// TwinCAT 3 PLC project PLC_TMO_VAC
// Title: lcls-plc-tmo-vac
// Company: SLAC
// ProjectVersion: 0.0.0
// ProgramVersion: 3.1.4022.7
// libraries:
//   LCLS General, * (SLAC)
//   LCLS Vacuum, * (SLAC - LCLS)
//   LCLSVacuumSerialDriverLib, * (SLAC - LCLS)
//   PMPS, * (SLAC - LCLS)
//   Tc2_SerialCom, * (Beckhoff Automation GmbH)
//   Tc2_Standard, * (Beckhoff Automation GmbH)
//   Tc2_System, * (Beckhoff Automation GmbH)
//   Tc3_Module, * (Beckhoff Automation GmbH)
// project tree:
//   / ComTask.TcTTO (not stored), FSVTask.TcTTO (not stored), PlcTask.TcTTO (not stored)
//   DUTs/ E_STATES.TcDUT (not stored)
//   GVLs/ GVL_COM.TcGVL (not stored), GVL_FEE_Device.TcGVL (not stored), GVL_FSV_PMPS.TcGVL, GVL_FS_Devices.TcGVL (not stored), GVL_Hutch_Gauges.TcGVL (not stored), GVL_Hutch_Pumps.TcGVL (not stored), GVL_Hutch_Valves.TcGVL (not stored), GVL_IP1_ECAT.TcGVL (not stored), GVL_PMPS.TcGVL, GVL_Variables.TcGVL
//   POUs/ DIAGNOSTICS.TcPOU (not stored), FB_VRC_NO_FFO_VLS.TcPOU (not stored), F_Turbo_Protection_ILK.TcPOU (not stored), MAIN.TcPOU, PRG_HV_SAFETY.TcPOU (not stored), PRG_PMPS.TcPOU, PRG_Hutch_Ion_Pumps.TcPOU (not stored), PRG_COM.TcPOU (not stored), PRG_FEE.TcPOU (not stored), PRG_FSV.TcPOU (not stored), PRG_FSV_Interfaces.TcPOU (not stored), PRG_Hutch_Beamline_Valves.TcPOU, PRG_Hutch_Gauges.TcPOU (not stored), PRG_IP1_ECAT_Interfaces.TcPOU (not stored), PRG_Roughing_Pumps.TcPOU, PRG_Section_2.TcPOU (not stored)
// real-time tasks:
//   TASK PlcTask: cycle T#10ms, priority 20, ADS port 350
//   TASK ComTask: cycle T#11ms, priority 30, ADS port 351
//   TASK FSVTask: cycle T#2ms, priority 15, ADS port 352
// I/O:
//   DEVICE Device 1 (EtherCAT)
// variable links:
//   PLC_TMO_VAC Instance <-> Device 1 (EtherCAT)/B940-R20-CX0 (EK1200)/CX0_E1 (EL2202)
//     ComTask Outputs/GVL_PMPS.g_FastFaultOutput1.q_xFastFaultOut <-> Channel 1/Output
//     ComTask Outputs/GVL_PMPS.g_FastFaultOutput2.q_xFastFaultOut <-> Channel 2/Output
//   PLC_TMO_VAC Instance <-> Device 1 (EtherCAT)/B940-R20-CX0 (EK1200)/CX0_E10_QPC2 (EL1004)
//     ComTask Inputs/GVL_FEE_Device.PC4K4_XTES_PIP_01.i_xSP_DI <-> Channel 1/Input
//     ComTask Inputs/GVL_FEE_Device.TV1K4_PIP_01.i_xSP_DI <-> Channel 3/Input
//     ComTask Inputs/GVL_Hutch_Pumps.MR2K4_KBO_PIP_01.i_xSP_DI <-> Channel 2/Input
//     ComTask Inputs/GVL_Hutch_Pumps.MR4K4_KBO_PIP_01.i_xSP_DI <-> Channel 4/Input
//   PLC_TMO_VAC Instance <-> Device 1 (EtherCAT)/B940-R20-CX0 (EK1200)/CX0_E11_QPC2 (EL2794)
//     ComTask Outputs/GVL_FEE_Device.PC4K4_XTES_PIP_01.q_xHVEna_DO <-> Channel 1/Output
//     ComTask Outputs/GVL_FEE_Device.TV1K4_PIP_01.q_xHVEna_DO <-> Channel 3/Output
//     ComTask Outputs/GVL_Hutch_Pumps.MR2K4_KBO_PIP_01.q_xHVEna_DO <-> Channel 2/Output
//     ComTask Outputs/GVL_Hutch_Pumps.MR4K4_KBO_PIP_01.q_xHVEna_DO <-> Channel 4/Output
//   PLC_TMO_VAC Instance <-> Device 1 (EtherCAT)/B940-R20-CX0 (EK1200)/CX0_E13 (EK1122)/IP1_ECAT (EL6692)
//     ComTask Inputs/GVL_IP1_ECAT.IP1_HV_SAFETY_ENABLE <-> IO Inputs/IP1_HV_SAFETY_ENABLE
//     ComTask Inputs/GVL_IP1_ECAT.IP1_MAIN_GAUGE.i_rPRESS <-> IO Inputs/IP1_MAIN_rPRESS
//     ComTask Inputs/GVL_IP1_ECAT.IP1_MAIN_GAUGE.i_xAT_VAC <-> IO Inputs/IP1_MAIN_xAT_VAC
//     ComTask Inputs/GVL_IP1_ECAT.IP1_MAIN_GAUGE.i_xPRESS_OK <-> IO Inputs/IP1_MAIN_xPRESS_OK
//     ComTask Inputs/GVL_IP1_ECAT.IP1_PLC_NAME <-> IO Inputs/ENDSTATION_PLC_NAME
//     ComTask Inputs/GVL_IP1_ECAT.IP1_ROUGH_VRC_01_AtOpnLS <-> IO Inputs/IP1_ROUGH_VRC_01_OPEN_LS
//     ComTask Inputs/GVL_IP1_ECAT.IP1_ROUGH_VRC_02_AtOpnLS <-> IO Inputs/IP1_ROUGH_VRC_02_OPEN_LS
//     ComTask Inputs/GVL_IP1_ECAT.IP1_ROUGH_VRC_03_AtOpnLS <-> IO Inputs/IP1_ROUGH_VRC_03_OPEN_LS
//     ComTask Inputs/GVL_IP1_ECAT.IP1_TURBOS_ALL_AtSpd <-> IO Inputs/IP1_TURBOS_ALL_AtSpd
//     ComTask Inputs/GVL_IP1_ECAT.xEcatBridge_External_device_not_connected <-> SYNC Inputs/External device not connected
//     ComTask Inputs/GVL_IP1_ECAT.xEcatBridge_TxPDO_state <-> SYNC Inputs/TxPDO state
//     ComTask Inputs/GVL_IP1_ECAT.xEcatBridge_WcState <-> WcState/WcState
//     ComTask Outputs/GVL_IP1_ECAT.My_PLC_NAME <-> IO Outputs/HUTCH_PLC_NAME
//     ComTask Outputs/GVL_IP1_ECAT.ROUGH1_VRC_01_AtOpnLS <-> IO Outputs/TMO_ROUGH1_VRC_01_OPEN_LS
//     ComTask Outputs/GVL_IP1_ECAT.ROUGH2_VRC_01_AtOpnLS <-> IO Outputs/TMO_ROUGH2_VRC_01_OPEN_LS
//   PLC_TMO_VAC Instance <-> Device 1 (EtherCAT)/B940-R20-CX0 (EK1200)/CX0_E1A (EL2202)
//     FSVTask Outputs/GVL_PMPS.g_FastFaultOutput3.q_xFastFaultOut <-> Channel 1/Output
//     FSVTask Outputs/GVL_PMPS.g_FastFaultOutput4.q_xFastFaultOut <-> Channel 2/Output
//   PLC_TMO_VAC Instance <-> Device 1 (EtherCAT)/B940-R20-CX0 (EK1200)/CX0_E2_EXILK (EL1008)
//     ComTask Inputs/GVL_FEE_Device.USVacOk_HI <-> Channel 1/Input
//     ComTask Inputs/GVL_FEE_Device.USVacOk_LO <-> Channel 3/Input
//   PLC_TMO_VAC Instance <-> Device 1 (EtherCAT)/B940-R20-CX0 (EK1200)/CX0_E6_QPC1 (EL3064)
//     ComTask Inputs/GVL_FEE_Device.MR1K4_SOMS_PIP_01.i_iPRESS <-> AI Standard Channel 1/Value
//     ComTask Inputs/GVL_FEE_Device.ST1K4_TEST_PIP_01.i_iPRESS <-> AI Standard Channel 2/Value
//     ComTask Inputs/GVL_FEE_Device.ST2K4_BCS_PIP_01.i_iPRESS <-> AI Standard Channel 3/Value
//     ComTask Inputs/GVL_FEE_Device.ST3K4_PPS_PIP_01.i_iPRESS <-> AI Standard Channel 4/Value
//   PLC_TMO_VAC Instance <-> Device 1 (EtherCAT)/B940-R20-CX0 (EK1200)/CX0_E7_QPC1 (EL1004)
//     ComTask Inputs/GVL_FEE_Device.MR1K4_SOMS_PIP_01.i_xSP_DI <-> Channel 1/Input
//     ComTask Inputs/GVL_FEE_Device.ST1K4_TEST_PIP_01.i_xSP_DI <-> Channel 2/Input
//     ComTask Inputs/GVL_FEE_Device.ST2K4_BCS_PIP_01.i_xSP_DI <-> Channel 3/Input
//     ComTask Inputs/GVL_FEE_Device.ST3K4_PPS_PIP_01.i_xSP_DI <-> Channel 4/Input
//   PLC_TMO_VAC Instance <-> Device 1 (EtherCAT)/B940-R20-CX0 (EK1200)/CX0_E8_QPC1 (EL2794)
//     ComTask Outputs/GVL_FEE_Device.MR1K4_SOMS_PIP_01.q_xHVEna_DO <-> Channel 1/Output
//     ComTask Outputs/GVL_FEE_Device.ST1K4_TEST_PIP_01.q_xHVEna_DO <-> Channel 2/Output
//     ComTask Outputs/GVL_FEE_Device.ST2K4_BCS_PIP_01.q_xHVEna_DO <-> Channel 3/Output
//     ComTask Outputs/GVL_FEE_Device.ST3K4_PPS_PIP_01.q_xHVEna_DO <-> Channel 4/Output
//   PLC_TMO_VAC Instance <-> Device 1 (EtherCAT)/B940-R20-CX0 (EK1200)/CX0_E9_QPC2 (EL3064)
//     ComTask Inputs/GVL_FEE_Device.PC4K4_XTES_PIP_01.i_iPRESS <-> AI Standard Channel 1/Value
//     ComTask Inputs/GVL_FEE_Device.TV1K4_PIP_01.i_iPRESS <-> AI Standard Channel 3/Value
//     ComTask Inputs/GVL_Hutch_Pumps.MR2K4_KBO_PIP_01.i_iPRESS <-> AI Standard Channel 2/Value
//     ComTask Inputs/GVL_Hutch_Pumps.MR4K4_KBO_PIP_01.i_iPRESS <-> AI Standard Channel 4/Value
//   PLC_TMO_VAC Instance <-> Device 1 (EtherCAT)/B940_K4S20_EB1  (EP2338-0002)
//     ComTask Inputs/GVL_FEE_Device.TV1K4_VGC_01.i_xClsLS <-> Channel 2/Input
//     ComTask Inputs/GVL_FEE_Device.TV1K4_VGC_02.i_xClsLS <-> Channel 6/Input
//     ComTask Inputs/GVL_FEE_Device.TV1K4_VGC_01.i_xOpnLS <-> Channel 1/Input
//     ComTask Inputs/GVL_FEE_Device.TV1K4_VGC_02.i_xOpnLS <-> Channel 5/Input
//     ComTask Outputs/GVL_FEE_Device.TV1K4_VGC_01.q_xOPN_DO <-> Channel 11/Output
//     ComTask Outputs/GVL_FEE_Device.TV1K4_VGC_02.q_xOPN_DO <-> Channel 15/Output
//   PLC_TMO_VAC Instance <-> Device 1 (EtherCAT)/B940_K4S20_EB2  (EP3174-0002)
//     ComTask Inputs/GVL_FEE_Device.TV1K4_GCC_01.i_iPRESS_R <-> AI Standard Channel 2/Value
//     ComTask Inputs/GVL_FEE_Device.TV1K4_GPI_01.i_iPRESS_R <-> AI Standard Channel 1/Value
//   PLC_TMO_VAC Instance <-> Device 1 (EtherCAT)/B940_K4S20_EB3 (EP2624-0002)
//     ComTask Outputs/GVL_FEE_Device.TV1K4_GCC_01.q_xHV_DIS <-> Channel 1/Output
//   PLC_TMO_VAC Instance <-> Device 1 (EtherCAT)/B940_K4S20_EK0  (EK1100)/K4S20-E1-FSV (EL1004)
//     FSVTask Inputs/GVL_FS_Devices.TV1K4_VFS_1.i_xClsLS <-> Channel 1/Input
//     FSVTask Inputs/GVL_FS_Devices.TV1K4_VFS_1.i_xOpnLS <-> Channel 2/Input
//   PLC_TMO_VAC Instance <-> Device 1 (EtherCAT)/B940_K4S20_EK0  (EK1100)/K4S20-E2-FSV (EL2202)
//     FSVTask Outputs/GVL_FS_Devices.TV1K4_VFS_1.q_xClose_A <-> Channel 1/Output
//     FSVTask Outputs/GVL_FS_Devices.TV1K4_VFS_1.q_xClose_B <-> Channel 2/Output
//   PLC_TMO_VAC Instance <-> Device 1 (EtherCAT)/B940_K4S20_EK0  (EK1100)/K4S20-E3-FSV (EL2202)
//     FSVTask Outputs/GVL_FS_Devices.TV1K4_VFS_1.q_xClose_C <-> Channel 1/Output
//     FSVTask Outputs/GVL_FS_Devices.TV1K4_VFS_1.q_xOPN_DO <-> Channel 2/Output
//   PLC_TMO_VAC Instance <-> Device 1 (EtherCAT)/B940_K4S24_EB1 (EP3174-0002)
//     ComTask Inputs/GVL_FEE_Device.ST1K4_TEST_GCC_01.i_iPRESS_R <-> AI Standard Channel 2/Value
//     ComTask Inputs/GVL_FEE_Device.ST1K4_TEST_GPI_01.i_iPRESS_R <-> AI Standard Channel 1/Value
//   PLC_TMO_VAC Instance <-> Device 1 (EtherCAT)/B940_K4S24_EB2 (EP2624-0002)
//     ComTask Outputs/GVL_FEE_Device.ST1K4_TEST_GCC_01.q_xHV_DIS <-> Channel 1/Output
//   PLC_TMO_VAC Instance <-> Device 1 (EtherCAT)/B940_K4S28_EB1 (EP3174-0002)
//     ComTask Inputs/GVL_FEE_Device.ST2K4_BCS_GCC_01.i_iPRESS_R <-> AI Standard Channel 2/Value
//     ComTask Inputs/GVL_FEE_Device.ST2K4_BCS_GPI_01.i_iPRESS_R <-> AI Standard Channel 1/Value
//   PLC_TMO_VAC Instance <-> Device 1 (EtherCAT)/B940_K4S28_EB2 (EP2624-0002)
//     ComTask Outputs/GVL_FEE_Device.ST2K4_BCS_GCC_01.q_xHV_DIS <-> Channel 1/Output
//   PLC_TMO_VAC Instance <-> Device 1 (EtherCAT)/B940_K4S33_EB1 (EP2338-0002)
//     ComTask Inputs/GVL_FEE_Device.ST3K4_PPS_VGC_01.i_xClsLS <-> Channel 2/Input
//     ComTask Inputs/GVL_FEE_Device.ST3K4_PPS_VGC_01.i_xOpnLS <-> Channel 1/Input
//     ComTask Outputs/GVL_FEE_Device.ST3K4_PPS_VGC_01.q_xOPN_DO <-> Channel 11/Output
//   PLC_TMO_VAC Instance <-> Device 1 (EtherCAT)/B940_K4S33_EB2 (EP3174-0002)
//     ComTask Inputs/GVL_FEE_Device.PC4K4_XTES_GCC_01.i_iPRESS_R <-> AI Standard Channel 2/Value
//     ComTask Inputs/GVL_FEE_Device.PC4K4_XTES_GPI_01.i_iPRESS_R <-> AI Standard Channel 1/Value
//   PLC_TMO_VAC Instance <-> Device 1 (EtherCAT)/B940_K4S33_EB3 (EP2624-0002)
//     ComTask Outputs/GVL_FEE_Device.PC4K4_XTES_GCC_01.q_xHV_DIS <-> Channel 1/Output
//   PLC_TMO_VAC Instance <-> Device 1 (EtherCAT)/B940_R20_EK0 (EK1100)/R20_EK0_E1_MKS937B (EL3064)
//     ComTask Inputs/GVL_Hutch_Gauges.LI2K4_IP1_GFS_01.i_iPRESS_R <-> AI Standard Channel 1/Value
//   PLC_TMO_VAC Instance <-> Device 1 (EtherCAT)/B940_R20_EK0 (EK1100)/R20_EK0_E3_MKS937B (EL2794)
//     ComTask Outputs/GVL_Hutch_Gauges.LI2K4_IP1_GFS_01.q_xHV_DIS <-> Channel 1/Output
//     ComTask Outputs/GVL_Hutch_Pumps.PA2K4_IP1_PIP_01.q_xHVEna_DO <-> Channel 4/Output
//   PLC_TMO_VAC Instance <-> Device 1 (EtherCAT)/B940_R20_EK0 (EK1100)/R20_EK0_E5_MKS937B (EL1124)
//     ComTask Inputs/GVL_Hutch_Pumps.PA2K4_IP1_PIP_01.i_xError <-> Channel 4/Input
//     ComTask Inputs/GVL_Hutch_Pumps.PA2K4_IP1_PIP_01.i_xIP_ON <-> Channel 3/Input
//     FSVTask Inputs/GVL_FS_Devices.MR3K4_KBO_VFS_1.i_xTrigger <-> Channel 1/Input
//     FSVTask Inputs/GVL_FS_Devices.MR4K4_KBO_VFS_1.i_xTrigger <-> Channel 1/Input
//     FSVTask Inputs/GVL_FS_Devices.TV1K4_VFS_1.i_xTrigger <-> Channel 1/Input
//   PLC_TMO_VAC Instance <-> Device 1 (EtherCAT)/B940_R20_EK0 (EK1100)/R20_EK0_SIP (EL3174-0002)
//     ComTask Inputs/GVL_Hutch_Pumps.PA2K4_IP1_PIP_01.i_iPRESS <-> AI Standard Channel 1/Value
//   PLC_TMO_VAC Instance <-> Device 1 (EtherCAT)/TMO_K4S2_ EP1 (EP4374-0002)
//     ComTask Inputs/GVL_Hutch_Gauges.TMO_ROUGH1_GPI_02.i_iPRESS_R <-> AI Inputs Channel 1/Value
//     ComTask Inputs/GVL_Hutch_Gauges.TMO_ROUGH2_GPI_02.i_iPRESS_R <-> AI Inputs Channel 2/Value
//     ComTask Outputs/GVL_Hutch_Valves.TMO_ROUGH1_VFV_02.q_iRawPosition <-> AO Outputs Channel 3/Analog output
//     ComTask Outputs/GVL_Hutch_Valves.TMO_ROUGH2_VFV_01.q_iRawPosition <-> AO Outputs Channel 4/Analog output
//   PLC_TMO_VAC Instance <-> Device 1 (EtherCAT)/TMO_K4S2_DRL_01 (EK1100)/K4S2_01_E1_VFS (EL1004)
//     FSVTask Inputs/GVL_FS_Devices.MR3K4_KBO_VFS_1.i_xClsLS <-> Channel 1/Input
//     FSVTask Inputs/GVL_FS_Devices.MR3K4_KBO_VFS_1.i_xOpnLS <-> Channel 2/Input
//   PLC_TMO_VAC Instance <-> Device 1 (EtherCAT)/TMO_K4S2_DRL_01 (EK1100)/K4S2_01_E3_VFS (EL2202)
//     FSVTask Outputs/GVL_FS_Devices.MR3K4_KBO_VFS_1.q_xClose_A <-> Channel 1/Output
//     FSVTask Outputs/GVL_FS_Devices.MR3K4_KBO_VFS_1.q_xClose_B <-> Channel 2/Output
//   PLC_TMO_VAC Instance <-> Device 1 (EtherCAT)/TMO_K4S2_DRL_01 (EK1100)/K4S2_01_E4_VFS (EL2202)
//     FSVTask Outputs/GVL_FS_Devices.MR3K4_KBO_VFS_1.q_xClose_C <-> Channel 1/Output
//     FSVTask Outputs/GVL_FS_Devices.MR3K4_KBO_VFS_1.q_xOPN_DO <-> Channel 2/Output
//   PLC_TMO_VAC Instance <-> Device 1 (EtherCAT)/TMO_K4S2_DRL_01 (EK1100)/K4S2_01_E5 (EL1004)
//     ComTask Inputs/GVL_Hutch_Valves.MR2K4_KBO_VWC_01.i_xClsLS <-> Channel 2/Input
//     ComTask Inputs/GVL_Hutch_Valves.MR3K4_KBO_VWC_01.i_xClsLS <-> Channel 4/Input
//     ComTask Inputs/GVL_Hutch_Valves.MR2K4_KBO_VWC_01.i_xOpnLS <-> Channel 1/Input
//     ComTask Inputs/GVL_Hutch_Valves.MR3K4_KBO_VWC_01.i_xOpnLS <-> Channel 3/Input
//   PLC_TMO_VAC Instance <-> Device 1 (EtherCAT)/TMO_K4S2_DRL_01 (EK1100)/K4S2_01_E6 (EL2004)
//     ComTask Outputs/GVL_Hutch_Valves.MR2K4_KBO_VWC_01.q_xOPN_DO <-> Channel 1/Output
//     ComTask Outputs/GVL_Hutch_Valves.MR3K4_KBO_VWC_01.q_xOPN_DO <-> Channel 2/Output
//   PLC_TMO_VAC Instance <-> Device 1 (EtherCAT)/TMO_K4S2_DRL_02 (EK1100)/K4S2_02_E1 (EL3174)
//     ComTask Inputs/GVL_Hutch_Gauges.MR2K4_KBO_GCC_01.i_iPRESS_R <-> AI Standard Channel 3/Value
//     ComTask Inputs/GVL_Hutch_Gauges.MR2K4_KBO_GPI_01.i_iPRESS_R <-> AI Standard Channel 2/Value
//     ComTask Inputs/GVL_Hutch_Gauges.PA1K4_IP1_GCC_01.i_iPRESS_R <-> AI Standard Channel 4/Value
//   PLC_TMO_VAC Instance <-> Device 1 (EtherCAT)/TMO_K4S2_DRL_02 (EK1100)/K4S2_02_E10 (EL6021)
//     ComTask Inputs/GVL_COM.K4S2_02_E10_stComIn/D[0] <-> COM TxPDO-Map Inputs/Data In 0
//     ComTask Inputs/GVL_COM.K4S2_02_E10_stComIn/D[10] <-> COM TxPDO-Map Inputs/Data In 10
//     ComTask Inputs/GVL_COM.K4S2_02_E10_stComIn/D[11] <-> COM TxPDO-Map Inputs/Data In 11
//     ComTask Inputs/GVL_COM.K4S2_02_E10_stComIn/D[12] <-> COM TxPDO-Map Inputs/Data In 12
//     ComTask Inputs/GVL_COM.K4S2_02_E10_stComIn/D[13] <-> COM TxPDO-Map Inputs/Data In 13
//     ComTask Inputs/GVL_COM.K4S2_02_E10_stComIn/D[14] <-> COM TxPDO-Map Inputs/Data In 14
//     ComTask Inputs/GVL_COM.K4S2_02_E10_stComIn/D[15] <-> COM TxPDO-Map Inputs/Data In 15
//     ComTask Inputs/GVL_COM.K4S2_02_E10_stComIn/D[16] <-> COM TxPDO-Map Inputs/Data In 16
//     ComTask Inputs/GVL_COM.K4S2_02_E10_stComIn/D[17] <-> COM TxPDO-Map Inputs/Data In 17
//     ComTask Inputs/GVL_COM.K4S2_02_E10_stComIn/D[18] <-> COM TxPDO-Map Inputs/Data In 18
//     ComTask Inputs/GVL_COM.K4S2_02_E10_stComIn/D[19] <-> COM TxPDO-Map Inputs/Data In 19
//     ComTask Inputs/GVL_COM.K4S2_02_E10_stComIn/D[1] <-> COM TxPDO-Map Inputs/Data In 1
//     ComTask Inputs/GVL_COM.K4S2_02_E10_stComIn/D[20] <-> COM TxPDO-Map Inputs/Data In 20
//     ComTask Inputs/GVL_COM.K4S2_02_E10_stComIn/D[21] <-> COM TxPDO-Map Inputs/Data In 21
//     ComTask Inputs/GVL_COM.K4S2_02_E10_stComIn/D[2] <-> COM TxPDO-Map Inputs/Data In 2
//     ComTask Inputs/GVL_COM.K4S2_02_E10_stComIn/D[3] <-> COM TxPDO-Map Inputs/Data In 3
//     ComTask Inputs/GVL_COM.K4S2_02_E10_stComIn/D[4] <-> COM TxPDO-Map Inputs/Data In 4
//     ComTask Inputs/GVL_COM.K4S2_02_E10_stComIn/D[5] <-> COM TxPDO-Map Inputs/Data In 5
//     ComTask Inputs/GVL_COM.K4S2_02_E10_stComIn/D[6] <-> COM TxPDO-Map Inputs/Data In 6
//     ComTask Inputs/GVL_COM.K4S2_02_E10_stComIn/D[7] <-> COM TxPDO-Map Inputs/Data In 7
//     ComTask Inputs/GVL_COM.K4S2_02_E10_stComIn/D[8] <-> COM TxPDO-Map Inputs/Data In 8
//     ComTask Inputs/GVL_COM.K4S2_02_E10_stComIn/D[9] <-> COM TxPDO-Map Inputs/Data In 9
//     ComTask Inputs/GVL_COM.K4S2_02_E10_stComIn/Status <-> COM TxPDO-Map Inputs/Status
//     ComTask Outputs/GVL_COM.K4S2_02_E10_stComOut/Ctrl <-> COM RxPDO-Map Outputs/Ctrl
//     ComTask Outputs/GVL_COM.K4S2_02_E10_stComOut/D[0] <-> COM RxPDO-Map Outputs/Data Out 0
//     ComTask Outputs/GVL_COM.K4S2_02_E10_stComOut/D[10] <-> COM RxPDO-Map Outputs/Data Out 10
//     ComTask Outputs/GVL_COM.K4S2_02_E10_stComOut/D[11] <-> COM RxPDO-Map Outputs/Data Out 11
//     ComTask Outputs/GVL_COM.K4S2_02_E10_stComOut/D[12] <-> COM RxPDO-Map Outputs/Data Out 12
//     ComTask Outputs/GVL_COM.K4S2_02_E10_stComOut/D[13] <-> COM RxPDO-Map Outputs/Data Out 13
//     ComTask Outputs/GVL_COM.K4S2_02_E10_stComOut/D[14] <-> COM RxPDO-Map Outputs/Data Out 14
//     ComTask Outputs/GVL_COM.K4S2_02_E10_stComOut/D[15] <-> COM RxPDO-Map Outputs/Data Out 15
//     ComTask Outputs/GVL_COM.K4S2_02_E10_stComOut/D[16] <-> COM RxPDO-Map Outputs/Data Out 16
//     ComTask Outputs/GVL_COM.K4S2_02_E10_stComOut/D[17] <-> COM RxPDO-Map Outputs/Data Out 17
//     ComTask Outputs/GVL_COM.K4S2_02_E10_stComOut/D[18] <-> COM RxPDO-Map Outputs/Data Out 18
//     ComTask Outputs/GVL_COM.K4S2_02_E10_stComOut/D[19] <-> COM RxPDO-Map Outputs/Data Out 19
//     ComTask Outputs/GVL_COM.K4S2_02_E10_stComOut/D[1] <-> COM RxPDO-Map Outputs/Data Out 1
//     ComTask Outputs/GVL_COM.K4S2_02_E10_stComOut/D[20] <-> COM RxPDO-Map Outputs/Data Out 20
//     ComTask Outputs/GVL_COM.K4S2_02_E10_stComOut/D[21] <-> COM RxPDO-Map Outputs/Data Out 21
//     ComTask Outputs/GVL_COM.K4S2_02_E10_stComOut/D[2] <-> COM RxPDO-Map Outputs/Data Out 2
//     ComTask Outputs/GVL_COM.K4S2_02_E10_stComOut/D[3] <-> COM RxPDO-Map Outputs/Data Out 3
//     ComTask Outputs/GVL_COM.K4S2_02_E10_stComOut/D[4] <-> COM RxPDO-Map Outputs/Data Out 4
//     ComTask Outputs/GVL_COM.K4S2_02_E10_stComOut/D[5] <-> COM RxPDO-Map Outputs/Data Out 5
//     ComTask Outputs/GVL_COM.K4S2_02_E10_stComOut/D[6] <-> COM RxPDO-Map Outputs/Data Out 6
//     ComTask Outputs/GVL_COM.K4S2_02_E10_stComOut/D[7] <-> COM RxPDO-Map Outputs/Data Out 7
//     ComTask Outputs/GVL_COM.K4S2_02_E10_stComOut/D[8] <-> COM RxPDO-Map Outputs/Data Out 8
//     ComTask Outputs/GVL_COM.K4S2_02_E10_stComOut/D[9] <-> COM RxPDO-Map Outputs/Data Out 9
//   PLC_TMO_VAC Instance <-> Device 1 (EtherCAT)/TMO_K4S2_DRL_02 (EK1100)/K4S2_02_E11 (EL1004)
//     ComTask Inputs/GVL_Hutch_Pumps.PA1K4_IP1_PTM_01.i_xAtSpd <-> Channel 2/Input
//     ComTask Inputs/GVL_Hutch_Pumps.PA1K4_IP1_PTM_02.i_xAtSpd <-> Channel 4/Input
//     ComTask Inputs/GVL_Hutch_Pumps.PA1K4_IP1_PTM_01.i_xFaultNC <-> Channel 1/Input
//     ComTask Inputs/GVL_Hutch_Pumps.PA1K4_IP1_PTM_02.i_xFaultNC <-> Channel 3/Input
//   PLC_TMO_VAC Instance <-> Device 1 (EtherCAT)/TMO_K4S2_DRL_02 (EK1100)/K4S2_02_E12 (EL2794)
//     ComTask Outputs/GVL_Hutch_Pumps.PA1K4_IP1_PTM_01.q_RunDO <-> Channel 1/Output
//     ComTask Outputs/GVL_Hutch_Pumps.PA1K4_IP1_PTM_02.q_RunDO <-> Channel 3/Output
//     ComTask Outputs/GVL_Hutch_Pumps.PA1K4_IP1_PTM_01.q_xReset <-> Channel 2/Output
//     ComTask Outputs/GVL_Hutch_Pumps.PA1K4_IP1_PTM_02.q_xReset <-> Channel 4/Output
//   PLC_TMO_VAC Instance <-> Device 1 (EtherCAT)/TMO_K4S2_DRL_02 (EK1100)/K4S2_02_E13 (EL1004)
//     ComTask Inputs/GVL_Hutch_Pumps.PA1K4_IP1_PTM_03.i_xAtSpd <-> Channel 2/Input
//     ComTask Inputs/GVL_Hutch_Pumps.PA1K4_IP1_PTM_03.i_xFaultNC <-> Channel 1/Input
//   PLC_TMO_VAC Instance <-> Device 1 (EtherCAT)/TMO_K4S2_DRL_02 (EK1100)/K4S2_02_E14 (EL2794)
//     ComTask Outputs/GVL_Hutch_Pumps.PA1K4_IP1_PTM_03.q_RunDO <-> Channel 1/Output
//     ComTask Outputs/GVL_Hutch_Pumps.PA1K4_IP1_PTM_03.q_xReset <-> Channel 2/Output
//   PLC_TMO_VAC Instance <-> Device 1 (EtherCAT)/TMO_K4S2_DRL_02 (EK1100)/K4S2_02_E15 (EL1004)
//     ComTask Inputs/GVL_Hutch_Pumps.IM4K4_PPM_PTM_01.i_xAtSpd <-> Channel 2/Input
//     ComTask Inputs/GVL_Hutch_Pumps.IM4K4_PPM_PTM_01.i_xFaultNC <-> Channel 1/Input
//     ComTask Inputs/GVL_Hutch_Pumps.LI1K4_IP1_PTM_01.i_xAtSpd <-> Channel 4/Input
//     ComTask Inputs/GVL_Hutch_Pumps.LI1K4_IP1_PTM_01.i_xFaultNC <-> Channel 3/Input
//   PLC_TMO_VAC Instance <-> Device 1 (EtherCAT)/TMO_K4S2_DRL_02 (EK1100)/K4S2_02_E16 (EL2794)
//     ComTask Outputs/GVL_Hutch_Pumps.IM4K4_PPM_PTM_01.q_RunDO <-> Channel 1/Output
//     ComTask Outputs/GVL_Hutch_Pumps.LI1K4_IP1_PTM_01.q_RunDO <-> Channel 2/Output
//   PLC_TMO_VAC Instance <-> Device 1 (EtherCAT)/TMO_K4S2_DRL_02 (EK1100)/K4S2_02_E17 (EL6001)
//     ComTask Inputs/GVL_COM.K4S2_02_E17_stComIn/D[0] <-> COM Inputs/Data In 0
//     ComTask Inputs/GVL_COM.K4S2_02_E17_stComIn/D[10] <-> COM Inputs/Data In 10
//     ComTask Inputs/GVL_COM.K4S2_02_E17_stComIn/D[11] <-> COM Inputs/Data In 11
//     ComTask Inputs/GVL_COM.K4S2_02_E17_stComIn/D[12] <-> COM Inputs/Data In 12
//     ComTask Inputs/GVL_COM.K4S2_02_E17_stComIn/D[13] <-> COM Inputs/Data In 13
//     ComTask Inputs/GVL_COM.K4S2_02_E17_stComIn/D[14] <-> COM Inputs/Data In 14
//     ComTask Inputs/GVL_COM.K4S2_02_E17_stComIn/D[15] <-> COM Inputs/Data In 15
//     ComTask Inputs/GVL_COM.K4S2_02_E17_stComIn/D[16] <-> COM Inputs/Data In 16
//     ComTask Inputs/GVL_COM.K4S2_02_E17_stComIn/D[17] <-> COM Inputs/Data In 17
//     ComTask Inputs/GVL_COM.K4S2_02_E17_stComIn/D[18] <-> COM Inputs/Data In 18
//     ComTask Inputs/GVL_COM.K4S2_02_E17_stComIn/D[19] <-> COM Inputs/Data In 19
//     ComTask Inputs/GVL_COM.K4S2_02_E17_stComIn/D[1] <-> COM Inputs/Data In 1
//     ComTask Inputs/GVL_COM.K4S2_02_E17_stComIn/D[20] <-> COM Inputs/Data In 20
//     ComTask Inputs/GVL_COM.K4S2_02_E17_stComIn/D[21] <-> COM Inputs/Data In 21
//     ComTask Inputs/GVL_COM.K4S2_02_E17_stComIn/D[2] <-> COM Inputs/Data In 2
//     ComTask Inputs/GVL_COM.K4S2_02_E17_stComIn/D[3] <-> COM Inputs/Data In 3
//     ComTask Inputs/GVL_COM.K4S2_02_E17_stComIn/D[4] <-> COM Inputs/Data In 4
//     ComTask Inputs/GVL_COM.K4S2_02_E17_stComIn/D[5] <-> COM Inputs/Data In 5
//     ComTask Inputs/GVL_COM.K4S2_02_E17_stComIn/D[6] <-> COM Inputs/Data In 6
//     ComTask Inputs/GVL_COM.K4S2_02_E17_stComIn/D[7] <-> COM Inputs/Data In 7
//     ComTask Inputs/GVL_COM.K4S2_02_E17_stComIn/D[8] <-> COM Inputs/Data In 8
//     ComTask Inputs/GVL_COM.K4S2_02_E17_stComIn/D[9] <-> COM Inputs/Data In 9
//     ComTask Inputs/GVL_COM.K4S2_02_E17_stComIn/Status <-> COM Inputs/Status
//     ComTask Outputs/GVL_COM.K4S2_02_E17_stComOut/Ctrl <-> COM Outputs/Ctrl
//     ComTask Outputs/GVL_COM.K4S2_02_E17_stComOut/D[0] <-> COM Outputs/Data Out 0
//     ComTask Outputs/GVL_COM.K4S2_02_E17_stComOut/D[10] <-> COM Outputs/Data Out 10
//     ComTask Outputs/GVL_COM.K4S2_02_E17_stComOut/D[11] <-> COM Outputs/Data Out 11
//     ComTask Outputs/GVL_COM.K4S2_02_E17_stComOut/D[12] <-> COM Outputs/Data Out 12
//     ComTask Outputs/GVL_COM.K4S2_02_E17_stComOut/D[13] <-> COM Outputs/Data Out 13
//     ComTask Outputs/GVL_COM.K4S2_02_E17_stComOut/D[14] <-> COM Outputs/Data Out 14
//     ComTask Outputs/GVL_COM.K4S2_02_E17_stComOut/D[15] <-> COM Outputs/Data Out 15
//     ComTask Outputs/GVL_COM.K4S2_02_E17_stComOut/D[16] <-> COM Outputs/Data Out 16
//     ComTask Outputs/GVL_COM.K4S2_02_E17_stComOut/D[17] <-> COM Outputs/Data Out 17
//     ComTask Outputs/GVL_COM.K4S2_02_E17_stComOut/D[18] <-> COM Outputs/Data Out 18
//     ComTask Outputs/GVL_COM.K4S2_02_E17_stComOut/D[19] <-> COM Outputs/Data Out 19
//     ComTask Outputs/GVL_COM.K4S2_02_E17_stComOut/D[1] <-> COM Outputs/Data Out 1
//     ComTask Outputs/GVL_COM.K4S2_02_E17_stComOut/D[20] <-> COM Outputs/Data Out 20
//     ComTask Outputs/GVL_COM.K4S2_02_E17_stComOut/D[21] <-> COM Outputs/Data Out 21
//     ComTask Outputs/GVL_COM.K4S2_02_E17_stComOut/D[2] <-> COM Outputs/Data Out 2
//     ComTask Outputs/GVL_COM.K4S2_02_E17_stComOut/D[3] <-> COM Outputs/Data Out 3
//     ComTask Outputs/GVL_COM.K4S2_02_E17_stComOut/D[4] <-> COM Outputs/Data Out 4
//     ComTask Outputs/GVL_COM.K4S2_02_E17_stComOut/D[5] <-> COM Outputs/Data Out 5
//     ComTask Outputs/GVL_COM.K4S2_02_E17_stComOut/D[6] <-> COM Outputs/Data Out 6
//     ComTask Outputs/GVL_COM.K4S2_02_E17_stComOut/D[7] <-> COM Outputs/Data Out 7
//     ComTask Outputs/GVL_COM.K4S2_02_E17_stComOut/D[8] <-> COM Outputs/Data Out 8
//     ComTask Outputs/GVL_COM.K4S2_02_E17_stComOut/D[9] <-> COM Outputs/Data Out 9
//   PLC_TMO_VAC Instance <-> Device 1 (EtherCAT)/TMO_K4S2_DRL_02 (EK1100)/K4S2_02_E18 (EL6001)
//     ComTask Inputs/GVL_COM.K4S2_02_E18_stComIn/D[0] <-> COM Inputs/Data In 0
//     ComTask Inputs/GVL_COM.K4S2_02_E18_stComIn/D[10] <-> COM Inputs/Data In 10
//     ComTask Inputs/GVL_COM.K4S2_02_E18_stComIn/D[11] <-> COM Inputs/Data In 11
//     ComTask Inputs/GVL_COM.K4S2_02_E18_stComIn/D[12] <-> COM Inputs/Data In 12
//     ComTask Inputs/GVL_COM.K4S2_02_E18_stComIn/D[13] <-> COM Inputs/Data In 13
//     ComTask Inputs/GVL_COM.K4S2_02_E18_stComIn/D[14] <-> COM Inputs/Data In 14
//     ComTask Inputs/GVL_COM.K4S2_02_E18_stComIn/D[15] <-> COM Inputs/Data In 15
//     ComTask Inputs/GVL_COM.K4S2_02_E18_stComIn/D[16] <-> COM Inputs/Data In 16
//     ComTask Inputs/GVL_COM.K4S2_02_E18_stComIn/D[17] <-> COM Inputs/Data In 17
//     ComTask Inputs/GVL_COM.K4S2_02_E18_stComIn/D[18] <-> COM Inputs/Data In 18
//     ComTask Inputs/GVL_COM.K4S2_02_E18_stComIn/D[19] <-> COM Inputs/Data In 19
//     ComTask Inputs/GVL_COM.K4S2_02_E18_stComIn/D[1] <-> COM Inputs/Data In 1
//     ComTask Inputs/GVL_COM.K4S2_02_E18_stComIn/D[20] <-> COM Inputs/Data In 20
//     ComTask Inputs/GVL_COM.K4S2_02_E18_stComIn/D[21] <-> COM Inputs/Data In 21
//     ComTask Inputs/GVL_COM.K4S2_02_E18_stComIn/D[2] <-> COM Inputs/Data In 2
//     ComTask Inputs/GVL_COM.K4S2_02_E18_stComIn/D[3] <-> COM Inputs/Data In 3
//     ComTask Inputs/GVL_COM.K4S2_02_E18_stComIn/D[4] <-> COM Inputs/Data In 4
//     ComTask Inputs/GVL_COM.K4S2_02_E18_stComIn/D[5] <-> COM Inputs/Data In 5
//     ComTask Inputs/GVL_COM.K4S2_02_E18_stComIn/D[6] <-> COM Inputs/Data In 6
//     ComTask Inputs/GVL_COM.K4S2_02_E18_stComIn/D[7] <-> COM Inputs/Data In 7
//     ComTask Inputs/GVL_COM.K4S2_02_E18_stComIn/D[8] <-> COM Inputs/Data In 8
//     ComTask Inputs/GVL_COM.K4S2_02_E18_stComIn/D[9] <-> COM Inputs/Data In 9
//     ComTask Inputs/GVL_COM.K4S2_02_E18_stComIn/Status <-> COM Inputs/Status
//     ComTask Outputs/GVL_COM.K4S2_02_E18_stComOut/Ctrl <-> COM Outputs/Ctrl
//     ComTask Outputs/GVL_COM.K4S2_02_E18_stComOut/D[0] <-> COM Outputs/Data Out 0
//     ComTask Outputs/GVL_COM.K4S2_02_E18_stComOut/D[10] <-> COM Outputs/Data Out 10
//     ComTask Outputs/GVL_COM.K4S2_02_E18_stComOut/D[11] <-> COM Outputs/Data Out 11
//     ComTask Outputs/GVL_COM.K4S2_02_E18_stComOut/D[12] <-> COM Outputs/Data Out 12
//     ComTask Outputs/GVL_COM.K4S2_02_E18_stComOut/D[13] <-> COM Outputs/Data Out 13
//     ComTask Outputs/GVL_COM.K4S2_02_E18_stComOut/D[14] <-> COM Outputs/Data Out 14
//     ComTask Outputs/GVL_COM.K4S2_02_E18_stComOut/D[15] <-> COM Outputs/Data Out 15
//     ComTask Outputs/GVL_COM.K4S2_02_E18_stComOut/D[16] <-> COM Outputs/Data Out 16
//     ComTask Outputs/GVL_COM.K4S2_02_E18_stComOut/D[17] <-> COM Outputs/Data Out 17
//     ComTask Outputs/GVL_COM.K4S2_02_E18_stComOut/D[18] <-> COM Outputs/Data Out 18
//     ComTask Outputs/GVL_COM.K4S2_02_E18_stComOut/D[19] <-> COM Outputs/Data Out 19
//     ComTask Outputs/GVL_COM.K4S2_02_E18_stComOut/D[1] <-> COM Outputs/Data Out 1
//     ComTask Outputs/GVL_COM.K4S2_02_E18_stComOut/D[20] <-> COM Outputs/Data Out 20
//     ComTask Outputs/GVL_COM.K4S2_02_E18_stComOut/D[21] <-> COM Outputs/Data Out 21
//     ComTask Outputs/GVL_COM.K4S2_02_E18_stComOut/D[2] <-> COM Outputs/Data Out 2
//     ComTask Outputs/GVL_COM.K4S2_02_E18_stComOut/D[3] <-> COM Outputs/Data Out 3
//     ComTask Outputs/GVL_COM.K4S2_02_E18_stComOut/D[4] <-> COM Outputs/Data Out 4
//     ComTask Outputs/GVL_COM.K4S2_02_E18_stComOut/D[5] <-> COM Outputs/Data Out 5
//     ComTask Outputs/GVL_COM.K4S2_02_E18_stComOut/D[6] <-> COM Outputs/Data Out 6
//     ComTask Outputs/GVL_COM.K4S2_02_E18_stComOut/D[7] <-> COM Outputs/Data Out 7
//     ComTask Outputs/GVL_COM.K4S2_02_E18_stComOut/D[8] <-> COM Outputs/Data Out 8
//     ComTask Outputs/GVL_COM.K4S2_02_E18_stComOut/D[9] <-> COM Outputs/Data Out 9
//   PLC_TMO_VAC Instance <-> Device 1 (EtherCAT)/TMO_K4S2_DRL_02 (EK1100)/K4S2_02_E19 (EL1004)
//     ComTask Inputs/GVL_Hutch_Valves.TMO_ROUGH1_VRC_01.i_xClsLS <-> Channel 2/Input
//     ComTask Inputs/GVL_Hutch_Valves.TMO_ROUGH2_VRC_01.i_xClsLS <-> Channel 4/Input
//     ComTask Inputs/GVL_Hutch_Valves.TMO_ROUGH1_VRC_01.i_xOpnLS <-> Channel 1/Input
//     ComTask Inputs/GVL_Hutch_Valves.TMO_ROUGH2_VRC_01.i_xOpnLS <-> Channel 3/Input
//   PLC_TMO_VAC Instance <-> Device 1 (EtherCAT)/TMO_K4S2_DRL_02 (EK1100)/K4S2_02_E2 (EL3174)
//     ComTask Inputs/GVL_Hutch_Gauges.IM4K4_PPM_GCC_01.i_iPRESS_R <-> AI Standard Channel 2/Value
//     ComTask Inputs/GVL_Hutch_Gauges.PA1K4_IP1_GPI_01.i_iPRESS_R <-> AI Standard Channel 1/Value
//   PLC_TMO_VAC Instance <-> Device 1 (EtherCAT)/TMO_K4S2_DRL_02 (EK1100)/K4S2_02_E20 (EL2004)
//     ComTask Outputs/GVL_Hutch_Valves.TMO_ROUGH1_VRC_01.q_xOPN_DO <-> Channel 1/Output
//     ComTask Outputs/GVL_Hutch_Valves.TMO_ROUGH2_VRC_01.q_xOPN_DO <-> Channel 2/Output
//     PlcTask Outputs/GVL_Variables.iHV_LOOP_FIM_ON <-> Channel 4/Output
//   PLC_TMO_VAC Instance <-> Device 1 (EtherCAT)/TMO_K4S2_DRL_02 (EK1100)/K4S2_02_E20A (EL1088)
//     ComTask Inputs/GVL_Hutch_Gauges.IM4K4_PPM_GCC_01.i_xHV_ON <-> Channel 1/Input
//   PLC_TMO_VAC Instance <-> Device 1 (EtherCAT)/TMO_K4S2_DRL_02 (EK1100)/K4S2_02_E5 (EL2624)
//     ComTask Outputs/GVL_Hutch_Gauges.IM4K4_PPM_GCC_01.q_xHV_DIS <-> Channel 4/Output
//     ComTask Outputs/GVL_Hutch_Gauges.MR2K4_KBO_GCC_01.q_xHV_DIS <-> Channel 2/Output
//     ComTask Outputs/GVL_Hutch_Gauges.PA1K4_IP1_GCC_01.q_xHV_DIS <-> Channel 3/Output
//   PLC_TMO_VAC Instance <-> Device 1 (EtherCAT)/TMO_K4S2_DRL_02 (EK1100)/K4S2_02_E7 (EL1124)
//     ComTask Inputs/GVL_Hutch_Gauges.MR2K4_KBO_GCC_01.i_xDisc_Active <-> Channel 4/Input
//     ComTask Inputs/GVL_Hutch_Gauges.MR2K4_KBO_GCC_01.i_xHV_ON <-> Channel 3/Input
//   PLC_TMO_VAC Instance <-> Device 1 (EtherCAT)/TMO_K4S2_DRL_02 (EK1100)/K4S2_02_E8 (EL1124)
//     ComTask Inputs/GVL_Hutch_Gauges.PA1K4_IP1_GCC_01.i_xDisc_Active <-> Channel 2/Input
//     ComTask Inputs/GVL_Hutch_Gauges.PA1K4_IP1_GCC_01.i_xHV_ON <-> Channel 1/Input
//   PLC_TMO_VAC Instance <-> Device 1 (EtherCAT)/TMO_K4S6_ EP1 (EP4374-0002)
//     ComTask Inputs/GVL_Hutch_Gauges.TMO_ROUGH1_GPI_03.i_iPRESS_R <-> AI Inputs Channel 1/Value
//     ComTask Outputs/GVL_Hutch_Valves.TMO_ROUGH1_VFV_03.q_iRawPosition <-> AO Outputs Channel 3/Analog output
//   PLC_TMO_VAC Instance <-> Device 1 (EtherCAT)/TMO_K4S6_DRL_01 (EK1100)/K4S6_01_E1 (EL1004)
//     ComTask Inputs/GVL_Hutch_Valves.TMO_ROUGH1_VRC_02.i_xClsLS <-> Channel 2/Input
//     ComTask Inputs/GVL_Hutch_Valves.TMO_ROUGH1_VRC_02.i_xOpnLS <-> Channel 1/Input
//   PLC_TMO_VAC Instance <-> Device 1 (EtherCAT)/TMO_K4S6_DRL_01 (EK1100)/K4S6_01_E11 (EL1004)
//     ComTask Inputs/GVL_Hutch_Pumps.IM5K4_PPM_PTM_01.i_xFaultNC <-> Channel 1/Input
//   PLC_TMO_VAC Instance <-> Device 1 (EtherCAT)/TMO_K4S6_DRL_01 (EK1100)/K4S6_01_E12 (EL2004)
//     ComTask Outputs/GVL_Hutch_Pumps.IM5K4_PPM_PTM_01.q_PumpingStation <-> Channel 1/Output
//   PLC_TMO_VAC Instance <-> Device 1 (EtherCAT)/TMO_K4S6_DRL_01 (EK1100)/K4S6_01_E14 (EL2624)
//     ComTask Outputs/GVL_Hutch_Gauges.IM5K4_PPM_GCC_01.q_xHV_DIS <-> Channel 2/Output
//     ComTask Outputs/GVL_Hutch_Gauges.MR4K4_KBO_GCC_01.q_xHV_DIS <-> Channel 4/Output
//     ComTask Outputs/GVL_Hutch_Gauges.PA2K4_IP1_GCC_01.q_xHV_DIS <-> Channel 3/Output
//     ComTask Outputs/GVL_Hutch_Gauges.TM1K4_GCC_01.q_xHV_DIS <-> Channel 1/Output
//   PLC_TMO_VAC Instance <-> Device 1 (EtherCAT)/TMO_K4S6_DRL_01 (EK1100)/K4S6_01_E15 (EL3174)
//     ComTask Inputs/GVL_Hutch_Gauges.IM5K4_PPM_GCC_01.i_iPRESS_R <-> AI Standard Channel 2/Value
//     ComTask Inputs/GVL_Hutch_Gauges.PA2K4_IP1_GCC_01.i_iPRESS_R <-> AI Standard Channel 3/Value
//     ComTask Inputs/GVL_Hutch_Gauges.PA2K4_IP1_GPI_01.i_iPRESS_R <-> AI Standard Channel 4/Value
//     ComTask Inputs/GVL_Hutch_Gauges.TM1K4_GCC_01.i_iPRESS_R <-> AI Standard Channel 1/Value
//   PLC_TMO_VAC Instance <-> Device 1 (EtherCAT)/TMO_K4S6_DRL_01 (EK1100)/K4S6_01_E18 (EL3174)
//     ComTask Inputs/GVL_Hutch_Gauges.MR4K4_KBO_GCC_01.i_iPRESS_R <-> AI Standard Channel 2/Value
//     ComTask Inputs/GVL_Hutch_Gauges.MR4K4_KBO_GPI_01.i_iPRESS_R <-> AI Standard Channel 1/Value
//   PLC_TMO_VAC Instance <-> Device 1 (EtherCAT)/TMO_K4S6_DRL_01 (EK1100)/K4S6_01_E2 (EL2004)
//     ComTask Outputs/GVL_Hutch_Valves.TMO_ROUGH1_VRC_02.q_xOPN_DO <-> Channel 1/Output
//   PLC_TMO_VAC Instance <-> Device 1 (EtherCAT)/TMO_K4S6_DRL_01 (EK1100)/K4S6_01_E20 (EL1124)
//     ComTask Inputs/GVL_Hutch_Gauges.IM5K4_PPM_GCC_01.i_xDisc_Active <-> Channel 4/Input
//     ComTask Inputs/GVL_Hutch_Gauges.IM5K4_PPM_GCC_01.i_xHV_ON <-> Channel 3/Input
//     ComTask Inputs/GVL_Hutch_Gauges.TM1K4_GCC_01.i_xDisc_Active <-> Channel 2/Input
//     ComTask Inputs/GVL_Hutch_Gauges.TM1K4_GCC_01.i_xHV_ON <-> Channel 1/Input
//   PLC_TMO_VAC Instance <-> Device 1 (EtherCAT)/TMO_K4S6_DRL_01 (EK1100)/K4S6_01_E21 (EL1124)
//     ComTask Inputs/GVL_Hutch_Gauges.MR4K4_KBO_GCC_01.i_xDisc_Active <-> Channel 4/Input
//     ComTask Inputs/GVL_Hutch_Gauges.MR4K4_KBO_GCC_01.i_xHV_ON <-> Channel 3/Input
//     ComTask Inputs/GVL_Hutch_Gauges.PA2K4_IP1_GCC_01.i_xDisc_Active <-> Channel 2/Input
//     ComTask Inputs/GVL_Hutch_Gauges.PA2K4_IP1_GCC_01.i_xHV_ON <-> Channel 1/Input
//   PLC_TMO_VAC Instance <-> Device 1 (EtherCAT)/TMO_K4S6_DRL_01 (EK1100)/K4S6_01_E3 (EL1004)
//     ComTask Inputs/GVL_Hutch_Valves.LI3K4_IP1_VWC_01.i_xClsLS <-> Channel 2/Input
//     ComTask Inputs/GVL_Hutch_Valves.LI3K4_IP1_VWC_01.i_xOpnLS <-> Channel 1/Input
//     ComTask Inputs/GVL_Hutch_Valves.PC5K4_VWC_01.i_xClsLS <-> Channel 4/Input
//     ComTask Inputs/GVL_Hutch_Valves.PC5K4_VWC_01.i_xOpnLS <-> Channel 3/Input
//   PLC_TMO_VAC Instance <-> Device 1 (EtherCAT)/TMO_K4S6_DRL_01 (EK1100)/K4S6_01_E4 (EL2004)
//     ComTask Outputs/GVL_Hutch_Valves.LI3K4_IP1_VWC_01.q_xOPN_DO <-> Channel 1/Output
//     ComTask Outputs/GVL_Hutch_Valves.PC5K4_VWC_01.q_xOPN_DO <-> Channel 2/Output
//   PLC_TMO_VAC Instance <-> Device 1 (EtherCAT)/TMO_K4S6_DRL_01 (EK1100)/K4S6_01_E5 (EL6021)
//     ComTask Inputs/GVL_COM.K4S6_01_E5_stComIn/D[0] <-> COM TxPDO-Map Inputs/Data In 0
//     ComTask Inputs/GVL_COM.K4S6_01_E5_stComIn/D[10] <-> COM TxPDO-Map Inputs/Data In 10
//     ComTask Inputs/GVL_COM.K4S6_01_E5_stComIn/D[11] <-> COM TxPDO-Map Inputs/Data In 11
//     ComTask Inputs/GVL_COM.K4S6_01_E5_stComIn/D[12] <-> COM TxPDO-Map Inputs/Data In 12
//     ComTask Inputs/GVL_COM.K4S6_01_E5_stComIn/D[13] <-> COM TxPDO-Map Inputs/Data In 13
//     ComTask Inputs/GVL_COM.K4S6_01_E5_stComIn/D[14] <-> COM TxPDO-Map Inputs/Data In 14
//     ComTask Inputs/GVL_COM.K4S6_01_E5_stComIn/D[15] <-> COM TxPDO-Map Inputs/Data In 15
//     ComTask Inputs/GVL_COM.K4S6_01_E5_stComIn/D[16] <-> COM TxPDO-Map Inputs/Data In 16
//     ComTask Inputs/GVL_COM.K4S6_01_E5_stComIn/D[17] <-> COM TxPDO-Map Inputs/Data In 17
//     ComTask Inputs/GVL_COM.K4S6_01_E5_stComIn/D[18] <-> COM TxPDO-Map Inputs/Data In 18
//     ComTask Inputs/GVL_COM.K4S6_01_E5_stComIn/D[19] <-> COM TxPDO-Map Inputs/Data In 19
//     ComTask Inputs/GVL_COM.K4S6_01_E5_stComIn/D[1] <-> COM TxPDO-Map Inputs/Data In 1
//     ComTask Inputs/GVL_COM.K4S6_01_E5_stComIn/D[20] <-> COM TxPDO-Map Inputs/Data In 20
//     ComTask Inputs/GVL_COM.K4S6_01_E5_stComIn/D[21] <-> COM TxPDO-Map Inputs/Data In 21
//     ComTask Inputs/GVL_COM.K4S6_01_E5_stComIn/D[2] <-> COM TxPDO-Map Inputs/Data In 2
//     ComTask Inputs/GVL_COM.K4S6_01_E5_stComIn/D[3] <-> COM TxPDO-Map Inputs/Data In 3
//     ComTask Inputs/GVL_COM.K4S6_01_E5_stComIn/D[4] <-> COM TxPDO-Map Inputs/Data In 4
//     ComTask Inputs/GVL_COM.K4S6_01_E5_stComIn/D[5] <-> COM TxPDO-Map Inputs/Data In 5
//     ComTask Inputs/GVL_COM.K4S6_01_E5_stComIn/D[6] <-> COM TxPDO-Map Inputs/Data In 6
//     ComTask Inputs/GVL_COM.K4S6_01_E5_stComIn/D[7] <-> COM TxPDO-Map Inputs/Data In 7
//     ComTask Inputs/GVL_COM.K4S6_01_E5_stComIn/D[8] <-> COM TxPDO-Map Inputs/Data In 8
//     ComTask Inputs/GVL_COM.K4S6_01_E5_stComIn/D[9] <-> COM TxPDO-Map Inputs/Data In 9
//     ComTask Inputs/GVL_COM.K4S6_01_E5_stComIn/Status <-> COM TxPDO-Map Inputs/Status
//     ComTask Outputs/GVL_COM.K4S6_01_E5_stComOut/Ctrl <-> COM RxPDO-Map Outputs/Ctrl
//     ComTask Outputs/GVL_COM.K4S6_01_E5_stComOut/D[0] <-> COM RxPDO-Map Outputs/Data Out 0
//     ComTask Outputs/GVL_COM.K4S6_01_E5_stComOut/D[10] <-> COM RxPDO-Map Outputs/Data Out 10
//     ComTask Outputs/GVL_COM.K4S6_01_E5_stComOut/D[11] <-> COM RxPDO-Map Outputs/Data Out 11
//     ComTask Outputs/GVL_COM.K4S6_01_E5_stComOut/D[12] <-> COM RxPDO-Map Outputs/Data Out 12
//     ComTask Outputs/GVL_COM.K4S6_01_E5_stComOut/D[13] <-> COM RxPDO-Map Outputs/Data Out 13
//     ComTask Outputs/GVL_COM.K4S6_01_E5_stComOut/D[14] <-> COM RxPDO-Map Outputs/Data Out 14
//     ComTask Outputs/GVL_COM.K4S6_01_E5_stComOut/D[15] <-> COM RxPDO-Map Outputs/Data Out 15
//     ComTask Outputs/GVL_COM.K4S6_01_E5_stComOut/D[16] <-> COM RxPDO-Map Outputs/Data Out 16
//     ComTask Outputs/GVL_COM.K4S6_01_E5_stComOut/D[17] <-> COM RxPDO-Map Outputs/Data Out 17
//     ComTask Outputs/GVL_COM.K4S6_01_E5_stComOut/D[18] <-> COM RxPDO-Map Outputs/Data Out 18
//     ComTask Outputs/GVL_COM.K4S6_01_E5_stComOut/D[19] <-> COM RxPDO-Map Outputs/Data Out 19
//     ComTask Outputs/GVL_COM.K4S6_01_E5_stComOut/D[1] <-> COM RxPDO-Map Outputs/Data Out 1
//     ComTask Outputs/GVL_COM.K4S6_01_E5_stComOut/D[20] <-> COM RxPDO-Map Outputs/Data Out 20
//     ComTask Outputs/GVL_COM.K4S6_01_E5_stComOut/D[21] <-> COM RxPDO-Map Outputs/Data Out 21
//     ComTask Outputs/GVL_COM.K4S6_01_E5_stComOut/D[2] <-> COM RxPDO-Map Outputs/Data Out 2
//     ComTask Outputs/GVL_COM.K4S6_01_E5_stComOut/D[3] <-> COM RxPDO-Map Outputs/Data Out 3
//     ComTask Outputs/GVL_COM.K4S6_01_E5_stComOut/D[4] <-> COM RxPDO-Map Outputs/Data Out 4
//     ComTask Outputs/GVL_COM.K4S6_01_E5_stComOut/D[5] <-> COM RxPDO-Map Outputs/Data Out 5
//     ComTask Outputs/GVL_COM.K4S6_01_E5_stComOut/D[6] <-> COM RxPDO-Map Outputs/Data Out 6
//     ComTask Outputs/GVL_COM.K4S6_01_E5_stComOut/D[7] <-> COM RxPDO-Map Outputs/Data Out 7
//     ComTask Outputs/GVL_COM.K4S6_01_E5_stComOut/D[8] <-> COM RxPDO-Map Outputs/Data Out 8
//     ComTask Outputs/GVL_COM.K4S6_01_E5_stComOut/D[9] <-> COM RxPDO-Map Outputs/Data Out 9
//   PLC_TMO_VAC Instance <-> Device 1 (EtherCAT)/TMO_K4S6_DRL_01 (EK1100)/K4S6_01_E6 (EL1004)
//     ComTask Inputs/GVL_Hutch_Pumps.LI3K4_IP1_OUT_PTM_01.i_xAtSpd <-> Channel 1/Input
//     ComTask Inputs/GVL_Hutch_Pumps.LI3K4_IP1_OUT_PTM_01.i_xFaultNC <-> Channel 3/Input
//     ComTask Inputs/GVL_Hutch_Pumps.LI3K4_IP1_OUT_PTM_01.i_xRemote <-> Channel 2/Input
//     ComTask Inputs/GVL_Hutch_Pumps.TM1K4_PTM_01.i_xAtSpd <-> Channel 4/Input
//   PLC_TMO_VAC Instance <-> Device 1 (EtherCAT)/TMO_K4S6_DRL_01 (EK1100)/K4S6_01_E7 (EL2004)
//     ComTask Outputs/GVL_Hutch_Pumps.LI3K4_IP1_OUT_PTM_01.q_PumpingStation <-> Channel 3/Output
//     ComTask Outputs/GVL_Hutch_Pumps.LI3K4_IP1_OUT_PTM_01.q_RunDO <-> Channel 1/Output
//     ComTask Outputs/GVL_Hutch_Pumps.LI3K4_IP1_OUT_PTM_01.q_xRemote <-> Channel 2/Output
//     ComTask Outputs/GVL_Hutch_Pumps.TM1K4_PTM_01.q_RunDO <-> Channel 4/Output
//   PLC_TMO_VAC Instance <-> Device 1 (EtherCAT)/TMO_K4S6_DRL_01 (EK1100)/K4S6_01_E8 (EL1004)
//     ComTask Inputs/GVL_Hutch_Pumps.IM5K4_PPM_PTM_01.i_xAtSpd <-> Channel 3/Input
//     ComTask Inputs/GVL_Hutch_Pumps.IM5K4_PPM_PTM_01.i_xRemote <-> Channel 4/Input
//     ComTask Inputs/GVL_Hutch_Pumps.TM1K4_PTM_01.i_xFaultNC <-> Channel 2/Input
//     ComTask Inputs/GVL_Hutch_Pumps.TM1K4_PTM_01.i_xRemote <-> Channel 1/Input
//   PLC_TMO_VAC Instance <-> Device 1 (EtherCAT)/TMO_K4S6_DRL_01 (EK1100)/K4S6_01_E9 (EL2004)
//     ComTask Outputs/GVL_Hutch_Pumps.IM5K4_PPM_PTM_01.q_RunDO <-> Channel 3/Output
//     ComTask Outputs/GVL_Hutch_Pumps.IM5K4_PPM_PTM_01.q_xRemote <-> Channel 4/Output
//     ComTask Outputs/GVL_Hutch_Pumps.TM1K4_PTM_01.q_PumpingStation <-> Channel 2/Output
//     ComTask Outputs/GVL_Hutch_Pumps.TM1K4_PTM_01.q_xRemote <-> Channel 1/Output
//   PLC_TMO_VAC Instance <-> Device 1 (EtherCAT)/TMO_K4S8_DRL_01 (EK1100)/K4S8_01_E1 (EL1004)
//     FSVTask Inputs/GVL_FS_Devices.MR4K4_KBO_VFS_1.i_xClsLS <-> Channel 1/Input
//     FSVTask Inputs/GVL_FS_Devices.MR4K4_KBO_VFS_1.i_xOpnLS <-> Channel 2/Input
//   PLC_TMO_VAC Instance <-> Device 1 (EtherCAT)/TMO_K4S8_DRL_01 (EK1100)/K4S8_01_E3 (EL2202)
//     FSVTask Outputs/GVL_FS_Devices.MR4K4_KBO_VFS_1.q_xClose_A <-> Channel 1/Output
//     FSVTask Outputs/GVL_FS_Devices.MR4K4_KBO_VFS_1.q_xClose_B <-> Channel 2/Output
//   PLC_TMO_VAC Instance <-> Device 1 (EtherCAT)/TMO_K4S8_DRL_01 (EK1100)/K4S8_01_E4 (EL2202)
//     FSVTask Outputs/GVL_FS_Devices.MR4K4_KBO_VFS_1.q_xClose_C <-> Channel 1/Output
//     FSVTask Outputs/GVL_FS_Devices.MR4K4_KBO_VFS_1.q_xOPN_DO <-> Channel 2/Output
//   PLC_TMO_VAC Instance <-> Device 1 (EtherCAT)/TMO_K4S8_DRL_01 (EK1100)/K4S8_01_E5 (EL1004)
//     ComTask Inputs/GVL_Hutch_Valves.MR4K4_KBO_VWC_01.i_xClsLS <-> Channel 2/Input
//     ComTask Inputs/GVL_Hutch_Valves.MR5K4_KBO_VWC_01.i_xClsLS <-> Channel 4/Input
//     ComTask Inputs/GVL_Hutch_Valves.MR4K4_KBO_VWC_01.i_xOpnLS <-> Channel 1/Input
//     ComTask Inputs/GVL_Hutch_Valves.MR5K4_KBO_VWC_01.i_xOpnLS <-> Channel 3/Input
//   PLC_TMO_VAC Instance <-> Device 1 (EtherCAT)/TMO_K4S8_DRL_01 (EK1100)/K4S8_01_E6 (EL2004)
//     ComTask Outputs/GVL_Hutch_Valves.MR4K4_KBO_VWC_01.q_xOPN_DO <-> Channel 1/Output
//     ComTask Outputs/GVL_Hutch_Valves.MR5K4_KBO_VWC_01.q_xOPN_DO <-> Channel 2/Output
//   PLC_TMO_VAC Instance <-> Device 1 (EtherCAT)/TMO_K4S8_DRL_02 (EK1100)/K4S8_02_E1 (EL1004)
//     ComTask Inputs/GVL_Hutch_Valves.TM2K4_KBO_VWC_01.i_xClsLS <-> Channel 2/Input
//     ComTask Inputs/GVL_Hutch_Valves.TM2K4_KBO_VWC_01.i_xOpnLS <-> Channel 1/Input
//   PLC_TMO_VAC Instance <-> Device 1 (EtherCAT)/TMO_K4S8_DRL_02 (EK1100)/K4S8_02_E2 (EL2004)
//     ComTask Outputs/GVL_Hutch_Valves.TM2K4_KBO_VWC_01.q_xOPN_DO <-> Channel 1/Output
//   PLC_TMO_VAC Instance <-> Device 1 (EtherCAT)/TMO_K4S8_DRL_02 (EK1100)/K4S8_02_E3 (EL2624)
//     ComTask Outputs/GVL_Hutch_Gauges.PF2K4_WFS_GCC_01.q_xHV_DIS <-> Channel 2/Output
//     ComTask Outputs/GVL_Hutch_Gauges.TM2K4_KBO_GCC_01.q_xHV_DIS <-> Channel 1/Output
//   PLC_TMO_VAC Instance <-> Device 1 (EtherCAT)/TMO_K4S8_DRL_02 (EK1100)/K4S8_02_E4 (EL3174)
//     ComTask Inputs/GVL_Hutch_Gauges.PF2K4_WFS_GCC_01.i_iPRESS_R <-> AI Standard Channel 2/Value
//     ComTask Inputs/GVL_Hutch_Gauges.TM2K4_KBO_GCC_01.i_iPRESS_R <-> AI Standard Channel 1/Value
//     ComTask Inputs/GVL_Hutch_Gauges.TM2K4_KBO_GPI_01.i_iPRESS_R <-> AI Standard Channel 3/Value
//   PLC_TMO_VAC Instance <-> Device 1 (EtherCAT)/TMO_K4S8_DRL_02 (EK1100)/K4S8_02_E6A (EL1084)
//     ComTask Inputs/GVL_Hutch_Gauges.PF2K4_WFS_GCC_01.i_xHV_ON <-> Channel 1/Input
//   PLC_TMO_VAC Instance <-> Device 1 (EtherCAT)/TMO_K4S8_DRL_02 (EK1100)/K4S8_02_E8 (EL1124)
//     ComTask Inputs/GVL_Hutch_Gauges.TM2K4_KBO_GCC_01.i_xDisc_Active <-> Channel 2/Input
//     ComTask Inputs/GVL_Hutch_Gauges.TM2K4_KBO_GCC_01.i_xHV_ON <-> Channel 1/Input
//   PLC_TMO_VAC Instance <-> Device 1 (EtherCAT)/TMO_WALL_WEST_EP01 (EP4374-0002)
//     ComTask Inputs/GVL_Hutch_Gauges.TMO_ROUGH1_GPI_01.i_iPRESS_R <-> AI Inputs Channel 1/Value
//     ComTask Inputs/GVL_Hutch_Gauges.TMO_ROUGH2_GPI_01.i_iPRESS_R <-> AI Inputs Channel 2/Value
//     ComTask Outputs/GVL_Hutch_Valves.TMO_ROUGH1_VFV_01.q_iRawPosition <-> AO Outputs Channel 3/Analog output
//   PLC_TMO_VAC Instance <-> PLC_TMO_VAC/PLC_TMO_VAC Instance
//     ComTask Inputs/GVL_FS_Devices.MR3K4_KBO_VFS_Interface.i_eVFS_State <-> FSVTask Outputs/GVL_FS_Devices.MR3K4_KBO_VFS_1.q_eVFS_State
//     ComTask Inputs/GVL_FS_Devices.MR4K4_KBO_VFS_Interface.i_eVFS_State <-> FSVTask Outputs/GVL_FS_Devices.MR4K4_KBO_VFS_1.q_eVFS_State
//     ComTask Inputs/GVL_FS_Devices.MR3K4_KBO_VFS_Interface.i_xMPS_OK <-> FSVTask Outputs/GVL_FS_Devices.MR3K4_KBO_VFS_1.q_xMPS_OK
//     ComTask Inputs/GVL_FS_Devices.MR4K4_KBO_VFS_Interface.i_xMPS_OK <-> FSVTask Outputs/GVL_FS_Devices.MR4K4_KBO_VFS_1.q_xMPS_OK
//     ComTask Inputs/GVL_FS_Devices.MR3K4_KBO_VFS_Interface.i_xTrigger <-> FSVTask Outputs/GVL_FS_Devices.MR3K4_KBO_VFS_1.q_xTrigger
//     ComTask Inputs/GVL_FS_Devices.MR4K4_KBO_VFS_Interface.i_xTrigger <-> FSVTask Outputs/GVL_FS_Devices.MR4K4_KBO_VFS_1.q_xTrigger
//     ComTask Inputs/GVL_FS_Devices.MR3K4_KBO_VFS_Interface.i_xVAC_FAULT_OK <-> FSVTask Outputs/GVL_FS_Devices.MR3K4_KBO_VFS_1.q_xVAC_FAULT_OK
//     ComTask Inputs/GVL_FS_Devices.MR4K4_KBO_VFS_Interface.i_xVAC_FAULT_OK <-> FSVTask Outputs/GVL_FS_Devices.MR4K4_KBO_VFS_1.q_xVAC_FAULT_OK
//     ComTask Inputs/GVL_FS_Devices.MR3K4_KBO_VFS_Interface.i_xVFS_Closed <-> FSVTask Outputs/GVL_FS_Devices.MR3K4_KBO_VFS_1.q_xVFS_Closed
//     ComTask Inputs/GVL_FS_Devices.MR4K4_KBO_VFS_Interface.i_xVFS_Closed <-> FSVTask Outputs/GVL_FS_Devices.MR4K4_KBO_VFS_1.q_xVFS_Closed
//     ComTask Inputs/GVL_FS_Devices.MR3K4_KBO_VFS_Interface.i_xVFS_Open <-> FSVTask Outputs/GVL_FS_Devices.MR3K4_KBO_VFS_1.q_xVFS_Open
//     ComTask Inputs/GVL_FS_Devices.MR4K4_KBO_VFS_Interface.i_xVFS_Open <-> FSVTask Outputs/GVL_FS_Devices.MR4K4_KBO_VFS_1.q_xVFS_Open
//     ComTask Inputs/GVL_FS_Devices.TV1K4_VFS_Interface.i_eVFS_State <-> FSVTask Outputs/GVL_FS_Devices.TV1K4_VFS_1.q_eVFS_State
//     ComTask Inputs/GVL_FS_Devices.TV1K4_VFS_Interface.i_xMPS_OK <-> FSVTask Outputs/GVL_FS_Devices.TV1K4_VFS_1.q_xMPS_OK
//     ComTask Inputs/GVL_FS_Devices.TV1K4_VFS_Interface.i_xTrigger <-> FSVTask Outputs/GVL_FS_Devices.TV1K4_VFS_1.q_xTrigger
//     ComTask Inputs/GVL_FS_Devices.TV1K4_VFS_Interface.i_xVAC_FAULT_OK <-> FSVTask Outputs/GVL_FS_Devices.TV1K4_VFS_1.q_xVAC_FAULT_OK
//     ComTask Inputs/GVL_FS_Devices.TV1K4_VFS_Interface.i_xVFS_Closed <-> FSVTask Outputs/GVL_FS_Devices.TV1K4_VFS_1.q_xVFS_Closed
//     ComTask Inputs/GVL_FS_Devices.TV1K4_VFS_Interface.i_xVFS_Open <-> FSVTask Outputs/GVL_FS_Devices.TV1K4_VFS_1.q_xVFS_Open
//     ComTask Outputs/GVL_FS_Devices.MR3K4_KBO_VFS_Interface.q_xCLS_SW <-> FSVTask Inputs/GVL_FS_Devices.MR3K4_KBO_VFS_1.i_xCLS_SW
//     ComTask Outputs/GVL_FS_Devices.MR4K4_KBO_VFS_Interface.q_xCLS_SW <-> FSVTask Inputs/GVL_FS_Devices.MR4K4_KBO_VFS_1.i_xCLS_SW
//     ComTask Outputs/GVL_FS_Devices.MR3K4_KBO_VFS_Interface.q_xOPN_SW <-> FSVTask Inputs/GVL_FS_Devices.MR3K4_KBO_VFS_1.i_xOPN_SW
//     ComTask Outputs/GVL_FS_Devices.MR4K4_KBO_VFS_Interface.q_xOPN_SW <-> FSVTask Inputs/GVL_FS_Devices.MR4K4_KBO_VFS_1.i_xOPN_SW
//     ComTask Outputs/GVL_FS_Devices.MR3K4_KBO_VFS_Interface.q_xOverrideMode <-> FSVTask Inputs/GVL_FS_Devices.MR3K4_KBO_VFS_1.i_xOverrideMode
//     ComTask Outputs/GVL_FS_Devices.MR4K4_KBO_VFS_Interface.q_xOverrideMode <-> FSVTask Inputs/GVL_FS_Devices.MR4K4_KBO_VFS_1.i_xOverrideMode
//     ComTask Outputs/GVL_FS_Devices.MR3K4_KBO_VFS_Interface.q_xOverrideOpen <-> FSVTask Inputs/GVL_FS_Devices.MR3K4_KBO_VFS_1.i_xOverrideOpen
//     ComTask Outputs/GVL_FS_Devices.MR4K4_KBO_VFS_Interface.q_xOverrideOpen <-> FSVTask Inputs/GVL_FS_Devices.MR4K4_KBO_VFS_1.i_xOverrideOpen
//     ComTask Outputs/GVL_FS_Devices.MR3K4_KBO_VFS_Interface.q_xPRESS_OK <-> FSVTask Inputs/GVL_FS_Devices.MR3K4_KBO_VFS_1.i_xPress_OK
//     ComTask Outputs/GVL_FS_Devices.MR4K4_KBO_VFS_Interface.q_xPRESS_OK <-> FSVTask Inputs/GVL_FS_Devices.MR4K4_KBO_VFS_1.i_xPress_OK
//     ComTask Outputs/GVL_FS_Devices.MR3K4_KBO_VFS_Interface.q_xVAC_FAULT_Reset <-> FSVTask Inputs/GVL_FS_Devices.MR3K4_KBO_VFS_1.i_xVAC_FAULT_Reset
//     ComTask Outputs/GVL_FS_Devices.MR4K4_KBO_VFS_Interface.q_xVAC_FAULT_Reset <-> FSVTask Inputs/GVL_FS_Devices.MR4K4_KBO_VFS_1.i_xVAC_FAULT_Reset
//     ComTask Outputs/GVL_FS_Devices.MR3K4_KBO_VFS_Interface.q_xVetoValveClosed <-> FSVTask Inputs/GVL_FS_Devices.MR3K4_KBO_VFS_1.i_xVetoValveClosed
//     ComTask Outputs/GVL_FS_Devices.MR4K4_KBO_VFS_Interface.q_xVetoValveClosed <-> FSVTask Inputs/GVL_FS_Devices.MR4K4_KBO_VFS_1.i_xVetoValveClosed
//     ComTask Outputs/GVL_FS_Devices.MR3K4_KBO_VFS_Interface.q_xVetoValveOpenDO <-> FSVTask Inputs/GVL_FS_Devices.MR3K4_KBO_VFS_1.i_xVetoValveOpenDO
//     ComTask Outputs/GVL_FS_Devices.MR4K4_KBO_VFS_Interface.q_xVetoValveOpenDO <-> FSVTask Inputs/GVL_FS_Devices.MR4K4_KBO_VFS_1.i_xVetoValveOpenDO
//     ComTask Outputs/GVL_FS_Devices.TV1K4_VFS_Interface.q_xCLS_SW <-> FSVTask Inputs/GVL_FS_Devices.TV1K4_VFS_1.i_xCLS_SW
//     ComTask Outputs/GVL_FS_Devices.TV1K4_VFS_Interface.q_xOPN_SW <-> FSVTask Inputs/GVL_FS_Devices.TV1K4_VFS_1.i_xOPN_SW
//     ComTask Outputs/GVL_FS_Devices.TV1K4_VFS_Interface.q_xOverrideMode <-> FSVTask Inputs/GVL_FS_Devices.TV1K4_VFS_1.i_xOverrideMode
//     ComTask Outputs/GVL_FS_Devices.TV1K4_VFS_Interface.q_xOverrideOpen <-> FSVTask Inputs/GVL_FS_Devices.TV1K4_VFS_1.i_xOverrideOpen
//     ComTask Outputs/GVL_FS_Devices.TV1K4_VFS_Interface.q_xPRESS_OK <-> FSVTask Inputs/GVL_FS_Devices.TV1K4_VFS_1.i_xPress_OK
//     ComTask Outputs/GVL_FS_Devices.TV1K4_VFS_Interface.q_xVAC_FAULT_Reset <-> FSVTask Inputs/GVL_FS_Devices.TV1K4_VFS_1.i_xVAC_FAULT_Reset
//     ComTask Outputs/GVL_FS_Devices.TV1K4_VFS_Interface.q_xVetoValveClosed <-> FSVTask Inputs/GVL_FS_Devices.TV1K4_VFS_1.i_xVetoValveClosed
//     ComTask Outputs/GVL_FS_Devices.TV1K4_VFS_Interface.q_xVetoValveOpenDO <-> FSVTask Inputs/GVL_FS_Devices.TV1K4_VFS_1.i_xVetoValveOpenDO
//     FSVTask Inputs/GVL_FS_Devices.MR3K4_KBO_VFS_1.i_xCLS_SW <-> ComTask Outputs/GVL_FS_Devices.MR3K4_KBO_VFS_Interface.q_xCLS_SW
//     FSVTask Inputs/GVL_FS_Devices.MR4K4_KBO_VFS_1.i_xCLS_SW <-> ComTask Outputs/GVL_FS_Devices.MR4K4_KBO_VFS_Interface.q_xCLS_SW
//     FSVTask Inputs/GVL_FS_Devices.MR3K4_KBO_VFS_1.i_xOPN_SW <-> ComTask Outputs/GVL_FS_Devices.MR3K4_KBO_VFS_Interface.q_xOPN_SW
//     FSVTask Inputs/GVL_FS_Devices.MR4K4_KBO_VFS_1.i_xOPN_SW <-> ComTask Outputs/GVL_FS_Devices.MR4K4_KBO_VFS_Interface.q_xOPN_SW
//     FSVTask Inputs/GVL_FS_Devices.MR3K4_KBO_VFS_1.i_xOverrideMode <-> ComTask Outputs/GVL_FS_Devices.MR3K4_KBO_VFS_Interface.q_xOverrideMode
//     FSVTask Inputs/GVL_FS_Devices.MR4K4_KBO_VFS_1.i_xOverrideMode <-> ComTask Outputs/GVL_FS_Devices.MR4K4_KBO_VFS_Interface.q_xOverrideMode
//     FSVTask Inputs/GVL_FS_Devices.MR3K4_KBO_VFS_1.i_xOverrideOpen <-> ComTask Outputs/GVL_FS_Devices.MR3K4_KBO_VFS_Interface.q_xOverrideOpen
//     FSVTask Inputs/GVL_FS_Devices.MR4K4_KBO_VFS_1.i_xOverrideOpen <-> ComTask Outputs/GVL_FS_Devices.MR4K4_KBO_VFS_Interface.q_xOverrideOpen
//     FSVTask Inputs/GVL_FS_Devices.MR3K4_KBO_VFS_1.i_xPress_OK <-> ComTask Outputs/GVL_FS_Devices.MR3K4_KBO_VFS_Interface.q_xPRESS_OK
//     FSVTask Inputs/GVL_FS_Devices.MR4K4_KBO_VFS_1.i_xPress_OK <-> ComTask Outputs/GVL_FS_Devices.MR4K4_KBO_VFS_Interface.q_xPRESS_OK
//     FSVTask Inputs/GVL_FS_Devices.MR3K4_KBO_VFS_1.i_xVAC_FAULT_Reset <-> ComTask Outputs/GVL_FS_Devices.MR3K4_KBO_VFS_Interface.q_xVAC_FAULT_Reset
//     FSVTask Inputs/GVL_FS_Devices.MR4K4_KBO_VFS_1.i_xVAC_FAULT_Reset <-> ComTask Outputs/GVL_FS_Devices.MR4K4_KBO_VFS_Interface.q_xVAC_FAULT_Reset
//     FSVTask Inputs/GVL_FS_Devices.MR3K4_KBO_VFS_1.i_xVetoValveClosed <-> ComTask Outputs/GVL_FS_Devices.MR3K4_KBO_VFS_Interface.q_xVetoValveClosed
//     FSVTask Inputs/GVL_FS_Devices.MR4K4_KBO_VFS_1.i_xVetoValveClosed <-> ComTask Outputs/GVL_FS_Devices.MR4K4_KBO_VFS_Interface.q_xVetoValveClosed
//     FSVTask Inputs/GVL_FS_Devices.MR3K4_KBO_VFS_1.i_xVetoValveOpenDO <-> ComTask Outputs/GVL_FS_Devices.MR3K4_KBO_VFS_Interface.q_xVetoValveOpenDO
//     FSVTask Inputs/GVL_FS_Devices.MR4K4_KBO_VFS_1.i_xVetoValveOpenDO <-> ComTask Outputs/GVL_FS_Devices.MR4K4_KBO_VFS_Interface.q_xVetoValveOpenDO
//     FSVTask Inputs/GVL_FS_Devices.TV1K4_VFS_1.i_xCLS_SW <-> ComTask Outputs/GVL_FS_Devices.TV1K4_VFS_Interface.q_xCLS_SW
//     FSVTask Inputs/GVL_FS_Devices.TV1K4_VFS_1.i_xOPN_SW <-> ComTask Outputs/GVL_FS_Devices.TV1K4_VFS_Interface.q_xOPN_SW
//     FSVTask Inputs/GVL_FS_Devices.TV1K4_VFS_1.i_xOverrideMode <-> ComTask Outputs/GVL_FS_Devices.TV1K4_VFS_Interface.q_xOverrideMode
//     FSVTask Inputs/GVL_FS_Devices.TV1K4_VFS_1.i_xOverrideOpen <-> ComTask Outputs/GVL_FS_Devices.TV1K4_VFS_Interface.q_xOverrideOpen
//     FSVTask Inputs/GVL_FS_Devices.TV1K4_VFS_1.i_xPress_OK <-> ComTask Outputs/GVL_FS_Devices.TV1K4_VFS_Interface.q_xPRESS_OK
//     FSVTask Inputs/GVL_FS_Devices.TV1K4_VFS_1.i_xVAC_FAULT_Reset <-> ComTask Outputs/GVL_FS_Devices.TV1K4_VFS_Interface.q_xVAC_FAULT_Reset
//     FSVTask Inputs/GVL_FS_Devices.TV1K4_VFS_1.i_xVetoValveClosed <-> ComTask Outputs/GVL_FS_Devices.TV1K4_VFS_Interface.q_xVetoValveClosed
//     FSVTask Inputs/GVL_FS_Devices.TV1K4_VFS_1.i_xVetoValveOpenDO <-> ComTask Outputs/GVL_FS_Devices.TV1K4_VFS_Interface.q_xVetoValveOpenDO
//     FSVTask Outputs/GVL_FS_Devices.MR3K4_KBO_VFS_1.q_eVFS_State <-> ComTask Inputs/GVL_FS_Devices.MR3K4_KBO_VFS_Interface.i_eVFS_State
//     FSVTask Outputs/GVL_FS_Devices.MR4K4_KBO_VFS_1.q_eVFS_State <-> ComTask Inputs/GVL_FS_Devices.MR4K4_KBO_VFS_Interface.i_eVFS_State
//     FSVTask Outputs/GVL_FS_Devices.MR3K4_KBO_VFS_1.q_xMPS_OK <-> ComTask Inputs/GVL_FS_Devices.MR3K4_KBO_VFS_Interface.i_xMPS_OK
//     FSVTask Outputs/GVL_FS_Devices.MR4K4_KBO_VFS_1.q_xMPS_OK <-> ComTask Inputs/GVL_FS_Devices.MR4K4_KBO_VFS_Interface.i_xMPS_OK
//     FSVTask Outputs/GVL_FS_Devices.MR3K4_KBO_VFS_1.q_xTrigger <-> ComTask Inputs/GVL_FS_Devices.MR3K4_KBO_VFS_Interface.i_xTrigger
//     FSVTask Outputs/GVL_FS_Devices.MR4K4_KBO_VFS_1.q_xTrigger <-> ComTask Inputs/GVL_FS_Devices.MR4K4_KBO_VFS_Interface.i_xTrigger
//     FSVTask Outputs/GVL_FS_Devices.MR3K4_KBO_VFS_1.q_xVAC_FAULT_OK <-> ComTask Inputs/GVL_FS_Devices.MR3K4_KBO_VFS_Interface.i_xVAC_FAULT_OK
//     FSVTask Outputs/GVL_FS_Devices.MR4K4_KBO_VFS_1.q_xVAC_FAULT_OK <-> ComTask Inputs/GVL_FS_Devices.MR4K4_KBO_VFS_Interface.i_xVAC_FAULT_OK
//     FSVTask Outputs/GVL_FS_Devices.MR3K4_KBO_VFS_1.q_xVFS_Closed <-> ComTask Inputs/GVL_FS_Devices.MR3K4_KBO_VFS_Interface.i_xVFS_Closed
//     FSVTask Outputs/GVL_FS_Devices.MR4K4_KBO_VFS_1.q_xVFS_Closed <-> ComTask Inputs/GVL_FS_Devices.MR4K4_KBO_VFS_Interface.i_xVFS_Closed
//     FSVTask Outputs/GVL_FS_Devices.MR3K4_KBO_VFS_1.q_xVFS_Open <-> ComTask Inputs/GVL_FS_Devices.MR3K4_KBO_VFS_Interface.i_xVFS_Open
//     FSVTask Outputs/GVL_FS_Devices.MR4K4_KBO_VFS_1.q_xVFS_Open <-> ComTask Inputs/GVL_FS_Devices.MR4K4_KBO_VFS_Interface.i_xVFS_Open
//     FSVTask Outputs/GVL_FS_Devices.TV1K4_VFS_1.q_eVFS_State <-> ComTask Inputs/GVL_FS_Devices.TV1K4_VFS_Interface.i_eVFS_State
//     FSVTask Outputs/GVL_FS_Devices.TV1K4_VFS_1.q_xMPS_OK <-> ComTask Inputs/GVL_FS_Devices.TV1K4_VFS_Interface.i_xMPS_OK
//     FSVTask Outputs/GVL_FS_Devices.TV1K4_VFS_1.q_xTrigger <-> ComTask Inputs/GVL_FS_Devices.TV1K4_VFS_Interface.i_xTrigger
//     FSVTask Outputs/GVL_FS_Devices.TV1K4_VFS_1.q_xVAC_FAULT_OK <-> ComTask Inputs/GVL_FS_Devices.TV1K4_VFS_Interface.i_xVAC_FAULT_OK
//     FSVTask Outputs/GVL_FS_Devices.TV1K4_VFS_1.q_xVFS_Closed <-> ComTask Inputs/GVL_FS_Devices.TV1K4_VFS_Interface.i_xVFS_Closed
//     FSVTask Outputs/GVL_FS_Devices.TV1K4_VFS_1.q_xVFS_Open <-> ComTask Inputs/GVL_FS_Devices.TV1K4_VFS_Interface.i_xVFS_Open

// ---- GVLs/GVL_FSV_PMPS.TcGVL
VAR_GLOBAL
(*
	
	{attribute 'pytmc' := 'pv: TMO:VAC:FFO:03  '}
   {attribute 'TcLinkTo' := '.q_xFastFaultOut:=TIIB[CX0_E1A (EL2202)]^Channel 1^Output'}
    g_FastFaultOutput3  :   FB_HardwareFFOutput;	//FFO for TV1K4-VFS-1
	
    {attribute 'pytmc' := 'pv: TMO:VAC:FFO:04  '}
   {attribute 'TcLinkTo' := '.q_xFastFaultOut:=TIIB[CX0_E1A (EL2202)]^Channel 2^Output'}
    g_FastFaultOutput4  :   FB_HardwareFFOutput;  // FF0 for MR3K4_KBO_VFS_01 & MR4K4_KBO_VFS_01
	
*)
END VAR

// ---- GVLs/GVL_PMPS.TcGVL
//{attribute 'qualified_only'}
VAR_GLOBAL
	
//Example implementation of the FFO
    {attribute 'pytmc' := 'pv: PLC:TMO:VAC:FFO:01    '}
    {attribute 'TcLinkTo' := '.q_xFastFaultOut:=TIIB[CX0_E1 (EL2202)]^Channel 1^Output'}
    g_FastFaultOutput1  :   FB_HardwareFFOutput:=(i_sNetID:='172.21.42.126.1.1');	//FFO for ST3K4_PPS's Upstream Components
	
	 {attribute 'pytmc' := 'pv: PLC:TMO:VAC:FFO:02  '}
    {attribute 'TcLinkTo' := '.q_xFastFaultOut:=TIIB[CX0_E1 (EL2202)]^Channel 2^Output'}
    g_FastFaultOutput2  :   FB_HardwareFFOutput:=(i_sNetID:='172.21.42.126.1.1');	//FFO for ST3K4_PPS's Downstream Components
	
	

	
	{attribute 'pytmc' := 'pv: TMO:VAC:FFO:03  '}
   {attribute 'TcLinkTo' := '.q_xFastFaultOut:=TIIB[CX0_E1A (EL2202)]^Channel 1^Output'}
    g_FastFaultOutput3  :   FB_HardwareFFOutput;	//FFO for TV1K4-VFS-1
	
    {attribute 'pytmc' := 'pv: TMO:VAC:FFO:04  '}
   {attribute 'TcLinkTo' := '.q_xFastFaultOut:=TIIB[CX0_E1A (EL2202)]^Channel 2^Output'}
    g_FastFaultOutput4  :   FB_HardwareFFOutput;  // FF0 for MR3K4_KBO_VFS_01 & MR4K4_KBO_VFS_01 
	
     {attribute 'pytmc' := 'pv: TMO:VAC:FFO:05  '}
	
	g_FastFaultOutput5 :    FB_HardwareFFOutput;  // FFO for ST4K4 photo terminator downstream devices


	
	{attribute 'pytmc' := '    pv: PLC:TMO:VAC:RESET:FF1    '}
	xReset_PMPS_FFO1	:	BOOL	:=	FALSE;		//FFO RESET for ST3K4_PPS's Upstream Components
	{attribute 'pytmc' := '    pv: PLC:TMO:VAC:RESET:FF2  '}
	xReset_PMPS_FFO2	:	BOOL	:=	FALSE;		//FFO RESET for ST3K4_PPS's Downstream Components
	{attribute 'pytmc' := '    pv: PLC:TMO:VAC:RESET:FF5  '}
	xReset_PMPS_FFO5	:	BOOL	:=	FALSE;		//FFO RESET for ST4K4_PPS's Downstream Components
	{attribute 'pytmc' := '        pv: PLC:TMO:VAC:ARB:01    '}
    g_fbArbiter1    :   FB_Arbiter(1); //Veto group downstream of MR1K1
	{attribute 'pytmc' := '        pv: PLC:TMO:VAC:ARB:02    '}
	g_fbArbiter2     :  FB_Arbiter(2);//Veto group downstream of ST3K4
	{attribute 'pytmc' := '        pv: PLC:TMO:VAC:ARB:03    '}
	g_fbArbiter3     :  FB_Arbiter(3);//Veto group downstream of ST4K4
	xTMO_FEE_MPS_OK: BOOL := TRUE;
	
	xTMO_NEH_MPS_OK: BOOL := TRUE;

END_VAR

// ---- GVLs/GVL_Variables.TcGVL
//{attribute 'qualified_only'}
VAR_GLOBAL


//	r_Accelerator_Setpoint	: REAL := 1E-12; (*unrealistic setpoint currently*)
    {attribute 'pytmc' := 'pv: TMO:FEE:VAC:OVRDON'}
    xSystemOverrideMode_FEE	: BOOL := FALSE; (* Global system override for the TMO FEE Vacuum System *)

    {attribute 'pytmc' := 'pv: TMO:NEH:VAC:OVRDON'}
    xSystemOverrideMode_TMO	: BOOL := FALSE; (* Global system override for the TMO hutch Vacuum System *)

    {attribute 'pytmc' := 'pv: TMO:NEH:TURBO:FAULT'}
    xTurboFault: BOOL := FALSE; (* True if any hutch turbo is not at speed or fault *)

    {attribute 'pytmc' := 'pv: TMO:NEH:VALVE:FAULT'}
    xBeamlineValveFault: BOOL := FALSE; (* True if any beamline valve is not open OK *)

        {attribute 'pytmc' := 'pv: TMO:NEH:ALL:GCC:ENABLE'}
    xGCC_Enable_SW: BOOL := FALSE; (* True if any hutch turbo is not at speed or fault *)

    {attribute 'pytmc' := 'pv: TMO:LAMP:PTM_NOK'}

    xLAMP_PTM_NOK AT%I*: BOOL := FALSE; (* True if any hutch turbo is not at speed or fault *)

    {attribute 'pytmc' := 'pv: TMO:VRC:DIFPRESS:BYPASS'}
    xBypassDiffPress_vrc1_vrc2 : BOOL;

    {attribute 'pytmc' := 'pv: TMO:FIM:HV_LOOP_PRESS'}
    iHV_LOOP_FIM_PRESSURE: REAL:= 8e-9;	//As Peter's request

    {attribute 'pytmc' := 'pv: TMO:FIM:HV_LOOP_ON'}
    {attribute 'TcLinkTo' := 'TIIB[K4S2_02_E20 (EL2004)]^Channel 4^Output'}
    iHV_LOOP_FIM_ON	AT %Q*: BOOL:= FALSE;

    {attribute 'pytmc' := 'pv: Pipe:replace:IP1'}
    xPipe_replace_IP1: BOOL := FALSE; (*tmo use piple to replace ip1 on  beamline*)

    {attribute 'pytmc' := 'pv: Psuedo:IP1:Gauge'}
    Psuedo_IP1_Gauge: ST_VG; //setup a psuedo gauge to select li2k4 instead of ip1 when pipe is in to replace ip1 08-21-25


END_VAR

// ---- POUs/MAIN.TcPOU
PROGRAM MAIN
VAR

	fbLogHandler : FB_LogHandler;
	
END_VAR


(* fbLogHandler();

(* FEE devices*)
PRG_FEE();
PRG_PMPS();
PRG_FSV_Interfaces();

(*  *)

(*Hutch*)
PRG_Hutch_Gauges();
PRG_Hutch_Beamline_Valves();
PRG_Roughing_Pumps();
PRG_Hutch_Ion_Pumps();

PRG_IP1_ECAT_Interfaces();    *)
PRG_HV_SAFETY();

END_PROGRAM

// ---- POUs/PRG_PMPS.TcPOU
PROGRAM PRG_PMPS
VAR
	fbArbiterIO : FB_SubSysToArbiter_IO;
	bRemove: BOOL;
	bRemove2: BOOL;
	bExist: BOOL;
	bExist2: BOOL;
	ID: UDINT;
	fb_VetoArbiter: FB_VetoArbiter;
	ff5_ff2_link_vac: FB_FastFault := (i_xAutoReset := TRUE, i_DevName := 'FF5 to FF2 Link', i_Desc := 'This is virtual FF5 fault, Please check ST4K4 downstream faulting device ', i_TypeCode := 16#9999);
	fb_VetoArbiter2: FB_VetoArbiter;
    
    bM1K1Veto : BOOL;
	bST3K4Veto : BOOL;
	bST4K4Veto : BOOL;
END_VAR


bM1K1Veto := NOT PMPS_GVL.stCurrentBeamParameters.aVetoDevices[PMPS.K_Stopper.MR1K1_OUT] 
                AND PMPS_GVL.stCurrentBeamParameters.aVetoDevices[PMPS.K_Stopper.MR1K1_IN];
bST3K4Veto := PMPS_GVL.stCurrentBeamParameters.aVetoDevices[PMPS.K_Stopper.ST3K4] OR bM1K1Veto;
bST4K4Veto := PMPS_GVL.stCurrentBeamParameters.aVetoDevices[PMPS.K_Stopper.ST4K4] OR bST3K4Veto;
(*FastFaultOuput*)
// Everything upstream ST3K4
g_FastFaultOutput1.Execute(i_xVeto:=bM1K1Veto, bAutoReset:= TRUE);

// Everything downstream of ST3K4
g_FastFaultOutput2.Execute(i_xVeto:=bST3K4Veto, bAutoReset:= TRUE);
// Everything downstream of ST4K4
g_FastFaultOutput5.Execute(i_xVeto:=bST4K4Veto, bAutoReset:= TRUE);
ff5_ff2_link_vac(
    io_fbFFHWO := GVL_PMPS.g_FastFaultOutput2,
    i_xOK := GVL_PMPS.g_FastFaultOutput5.q_xFastFaultOut);
	
// Preemptive system
//fbArbiterIO(Arbiter := g_fbArbiter1, fbFFHWO := g_FastFaultOutput1,
//	i_bVeto := bM1K1Veto);
    
//fb_VetoArbiter(bVeto:= PMPS_GVL.stCurrentBeamParameters.aVetoDevices[PMPS.K_Stopper.ST3K4],
//		HigherAuthority:=g_fbArbiter1 , 
	//	LowerAuthority:= g_fbArbiter2 , FFO:= g_FastFaultOutput2);
//fb_VetoArbiter2(bVeto:= PMPS_GVL.stCurrentBeamParameters.aVetoDevices[PMPS.K_Stopper.ST4K4], ??
//		HigherAuthority:=g_fbArbiter2 , 
//		LowerAuthority:= g_fbArbiter3 (*downstream of st4k4*), FFO:= g_FastFaultOutput5);

//Test and diagnostic stuff
bExist:= g_fbArbiter1.CheckRequestInPool(ID);
bExist2:= g_fbArbiter2.CheckRequestInPool(ID);
if (bRemove) THEN
	g_fbArbiter1.RemoveRequest(ID);
END_IF
if (bRemove2) THEN
	g_fbArbiter2.RemoveRequest(ID);
END_IF

END_PROGRAM

// ---- POUs/PRG_Hutch_Beamline_Valves.TcPOU
PROGRAM PRG_Hutch_Beamline_Valves
VAR
    LAMP_C2_GCC_01: FB_MKS500; // wrong. only need temporary before integrate with LAMP
    xAll_Turbo_isRunning : BOOL := False;


    ton_PA1K4_IP1_PTM_01_notRunning : TON;
    ton_PA1K4_IP1_PTM_02_notRunning : TON;
    ton_PA1K4_IP1_PTM_03_notRunning : TON;
    ton_IM4K4_PPM_PTM_01_notRunning : TON;
    ton_LI1K4_IP1_PTM_01_notRunning : TON;
    ton_LI3K4_IP1_OUT_PTM_01_notRunning : TON;
    ton_TM1K4_PTM_01_notRunning : TON;
    ton_IM5K4_PPM_PTM_01_notRunning : TON;

    tDelOK	:	TIME := T#30S;
    xExtIlkOK : BOOL;

    PA1K4_IP1_PTM_01_isRunning: BOOL;
    PA1K4_IP1_PTM_02_isRunning: BOOL;
    PA1K4_IP1_PTM_03_isRunning: BOOL;
    IM4K4_PPM_PTM_01_isRunning: BOOL;
    LI1K4_IP1_PTM_01_isRunning: BOOL;
    LI3K4_IP1_OUT_PTM_01_isRunning: BOOL;
    TM1K4_PTM_01_isRunning: BOOL;
    IM5K4_PPM_PTM_01_isRunning: BOOL;

    xValves_are_OPN_OK : BOOL;

END_VAR


(* Beamline window valves use VGC function. Valves allow to open when both upstream and downstream gauges
    reading pressure below than setpoints,  all turbo pumps are running and no faults, and all beamline valves
    in hutch are OPN_OK*)

(* check turbo pump status	*)
PA1K4_IP1_PTM_01_isRunning := PA1K4_IP1_PTM_01.iq_stPTM.eState = E_PumpState.pumpRUNNING;
ton_PA1K4_IP1_PTM_01_notRunning(IN:= NOT PA1K4_IP1_PTM_01_isRunning, PT:=tDelOK);

PA1K4_IP1_PTM_02_isRunning := PA1K4_IP1_PTM_02.iq_stPTM.eState = E_PumpState.pumpRUNNING;
ton_PA1K4_IP1_PTM_02_notRunning(IN:= NOT PA1K4_IP1_PTM_02_isRunning, PT:=tDelOK);

PA1K4_IP1_PTM_03_isRunning := PA1K4_IP1_PTM_03.iq_stPTM.eState = E_PumpState.pumpRUNNING;
ton_PA1K4_IP1_PTM_03_notRunning(IN:= NOT PA1K4_IP1_PTM_03_isRunning, PT:=tDelOK);

IM4K4_PPM_PTM_01_isRunning := IM4K4_PPM_PTM_01.iq_stPTM.eState = E_PumpState.pumpRUNNING;
ton_IM4K4_PPM_PTM_01_notRunning(IN:= NOT IM4K4_PPM_PTM_01_isRunning, PT:=tDelOK);

LI1K4_IP1_PTM_01_isRunning := LI1K4_IP1_PTM_01.iq_stPTM.eState = E_PumpState.pumpRUNNING;
ton_LI1K4_IP1_PTM_01_notRunning(IN:= NOT LI1K4_IP1_PTM_01_isRunning, PT:=tDelOK);

LI3K4_IP1_OUT_PTM_01_isRunning := LI3K4_IP1_OUT_PTM_01.iq_stPTM.eState = E_PumpState.pumpRUNNING;
ton_LI3K4_IP1_OUT_PTM_01_notRunning(IN:= NOT LI3K4_IP1_OUT_PTM_01_isRunning, PT:=tDelOK);

TM1K4_PTM_01_isRunning := TM1K4_PTM_01.iq_stPTM.eState = E_PumpState.pumpRUNNING;
ton_TM1K4_PTM_01_notRunning(IN:= NOT TM1K4_PTM_01_isRunning, PT:=tDelOK);

IM5K4_PPM_PTM_01_isRunning := IM5K4_PPM_PTM_01.iq_stPTM.eState = E_PumpState.pumpRUNNING;
ton_IM5K4_PPM_PTM_01_notRunning(IN:= NOT IM5K4_PPM_PTM_01_isRunning, PT:=tDelOK);

xTurboFault := ton_PA1K4_IP1_PTM_01_notRunning.Q OR ton_PA1K4_IP1_PTM_02_notRunning.Q OR
               ton_PA1K4_IP1_PTM_03_notRunning.Q OR ton_IM4K4_PPM_PTM_01_notRunning.Q OR
               ton_LI1K4_IP1_PTM_01_notRunning.Q OR ton_LI3K4_IP1_OUT_PTM_01_notRunning.Q OR
                ton_TM1K4_PTM_01_notRunning.Q OR ton_IM5K4_PPM_PTM_01_notRunning.Q
                OR NOT (IP1_TURBOS_ALL_AtSpd OR xPipe_replace_IP1); // add pipe to replace ip1 on 8-21-25

(* check beamline valve OPEN permit *)
(*xValves_are_OPN_OK :=  MR2K4_KBO_VWC_01.iq_stValve.xOPN_OK AND MR3K4_KBO_VWC_01.iq_stValve.xOPN_OK AND
                       LI3K4_IP1_VWC_01.iq_stValve.xOPN_OK AND PC5K4_VWC_01.iq_stValve.xOPN_OK ; *)

(*if not all beamline valves are OPN_OK, close all beamline valves*)
(*IF NOT xValves_are_OPN_OK Then
    MR2K4_KBO_VWC_01.M_Set_OPN_SW(false);
    MR3K4_KBO_VWC_01.M_Set_OPN_SW(false);
    LI3K4_IP1_VWC_01.M_Set_OPN_SW(false);
    PC5K4_VWC_01.M_Set_OPN_SW(false);
    xBeamlineValveFault := True;
ElSE
   xBeamlineValveFault := False;
END_IF
*)



MR2K4_KBO_VWC_01(
                i_stUSG := PC4K4_XTES_GCC_01.IG,
                i_stDSG:= MR2K4_KBO_GCC_01.IG,
                i_xDis_DPIlk := FALSE,
                i_xEPS_OK := TRUE,
                i_xPMPS_OK := TRUE ,
                i_xExt_OK := TRUE, // James request on Feb 2025
                i_xOverrideMode := xSystemOverrideMode_TMO,
                i_xReset := xReset_PMPS_FFO2,
                iq_stValve =>,
                io_fbFFHWO :=g_FastFaultOutput2,
                fbArbiter := g_fbArbiter2,
                i_nTransitionRootID := 47632,
                i_sDevName := 'MR2K4-KBO-VWC-01'

);


MR3K4_KBO_VWC_01(
                i_stUSG := MR2K4_KBO_GCC_01.IG,
                i_stDSG:= PA1K4_IP1_GCC_01.IG,
                i_xDis_DPIlk := FALSE,
                i_xEPS_OK := TRUE,
                i_xPMPS_OK := TRUE ,
                i_xExt_OK := NOT xTurboFault AND MR3K4_KBO_VFS_Interface.i_xVAC_FAULT_OK,
                i_xOverrideMode := xSystemOverrideMode_TMO,
                i_xReset := xReset_PMPS_FFO2,
                iq_stValve =>,
                io_fbFFHWO :=g_FastFaultOutput2,
                fbArbiter := g_fbArbiter2,
                i_nTransitionRootID := 47648,
                i_sDevName := 'MR3K4-KBO-VWC-01'

);
// setup a psuedo gauge to select li2k4 instead of ip1 when pipe is in to replace ip1 08-21-25
IF xPipe_replace_IP1 THEN
    Psuedo_IP1_Gauge := LI2K4_IP1_GFS_02.IG;
    Psuedo_IP1_Gauge.sPath := 'LI2K4_IP1_GFS_02';
ELSE
    Psuedo_IP1_Gauge := IP1_MAIN_GAUGE.VG;
    Psuedo_IP1_Gauge.sPath := 'IP1_MAIN_GAUGE';
END_IF
//add pipe in to replace ip1-08-21-25
LI3K4_IP1_VWC_01(
                i_stUSG := Psuedo_IP1_Gauge,
                i_stDSG:= IM5K4_PPM_GCC_01.IG,
                i_xDis_DPIlk := FALSE,
                i_xEPS_OK := TRUE,
                i_xPMPS_OK := TRUE ,
                i_xExt_OK := NOT xTurboFault,
                i_xOverrideMode := xSystemOverrideMode_TMO,
                i_xReset := xReset_PMPS_FFO2,
                iq_stValve =>,
                io_fbFFHWO :=g_FastFaultOutput2,
                fbArbiter := g_fbArbiter2,
                i_nTransitionRootID := 47664,
                i_sDevName := 'LI3K4-IP1-VWC-01'
);

PC5K4_VWC_01(
                i_stUSG := IM5K4_PPM_GCC_01.IG,
                i_stDSG:= PA2K4_IP1_GCC_01.IG,
                i_xDis_DPIlk := FALSE,
                i_xEPS_OK := TRUE,
                i_xPMPS_OK := TRUE,
                i_xExt_OK := NOT xTurboFault,
                i_xOverrideMode := xSystemOverrideMode_TMO,
                i_xReset := xReset_PMPS_FFO5,
                iq_stValve =>,
                io_fbFFHWO :=g_FastFaultOutput5,
                fbArbiter := g_fbArbiter3,
                i_nTransitionRootID := 47680,
                i_sDevName := 'PC5K4-VWC-01'
);

MR4K4_KBO_VWC_01(
                i_stUSG := PA2K4_IP1_GCC_01.IG,
                i_stDSG:= MR4K4_KBO_GCC_01.IG,
                i_xDis_DPIlk := FALSE,
                i_xEPS_OK := TRUE,
                i_xPMPS_OK := TRUE,
                i_xExt_OK := NOT xTurboFault,
                i_xOverrideMode := xSystemOverrideMode_TMO,
                i_xReset := xReset_PMPS_FFO2,
                iq_stValve =>,
                io_fbFFHWO :=g_FastFaultOutput5,
                fbArbiter := g_fbArbiter3,
                i_nTransitionRootID := 47696,
                i_sDevName := 'MR4K4-KBO-VWC-01'
);
// when dream arrives, this needs to be changes to dream gauge(downstream)
MR5K4_KBO_VWC_01(
                i_stUSG := MR4K4_KBO_GCC_01.IG,
                i_stDSG := stDreamMainGauge,
                i_xDis_DPIlk := FALSE,
                i_xEPS_OK := TRUE,
                i_xPMPS_OK := TRUE,
                i_xExt_OK := NOT xTurboFault,
                i_xOverrideMode := xSystemOverrideMode_TMO,
                i_xReset := xReset_PMPS_FFO2,
                iq_stValve =>,
                io_fbFFHWO :=g_FastFaultOutput5,
                fbArbiter := g_fbArbiter3,
                i_nTransitionRootID := 47697,
                i_sDevName := 'MR5K4-KBO-VWC-01'
);
//Currently there is no dream, so TM2K4 valve is always open during this configuration
TM2K4_KBO_VWC_01(
                i_stUSG := stDreamMainGauge,
                i_stDSG := TM2K4_KBO_GCC_01.IG,
                i_xDis_DPIlk := FALSE,
                i_xEPS_OK := TRUE,
                i_xPMPS_OK := TRUE,
                i_xExt_OK := NOT xTurboFault,
                i_xOverrideMode := xSystemOverrideMode_TMO,
                i_xReset := xReset_PMPS_FFO5,
                iq_stValve =>,
                io_fbFFHWO :=g_FastFaultOutput5,
                fbArbiter := g_fbArbiter3,
                i_nTransitionRootID := 47698,
                i_sDevName := 'TM2K4-KBO-VWC-01'
);

//VFV Valves James request to change on Feb 2025
TMO_ROUGH1_VFV_01(i_xExtIlkOK := FALSE);
TMO_ROUGH1_VFV_02(i_xExtIlkOK := TMO_ROUGH1_VRC_01.M_IsClosed() AND TMO_ROUGH2_VRC_01.M_IsClosed() AND MR3K4_KBO_VWC_01.M_IsClosed() AND LI3K4_IP1_VWC_01.M_IsClosed());
TMO_ROUGH1_VFV_03(i_xExtIlkOK := TMO_ROUGH1_VRC_02.M_IsClosed()AND MR3K4_KBO_VWC_01.M_IsClosed() AND LI3K4_IP1_VWC_01.M_IsClosed() AND PC5K4_VWC_01.M_IsClosed());
//TMO_ROUGH2_VFV_01(i_xExtIlkOK := TMO_ROUGH1_VRC_01.M_IsClosed() AND TMO_ROUGH2_VRC_01.M_IsClosed());
IF (IP1_ECAT_COM_ERROR OR xPipe_replace_IP1) THEN //If IP1 and Tmo beamline detect communication error,assuming IP1_ROUGH_VRC_02 open, tend to vent entire end station //add pipe in replacing ip1 8-21-25
    TMO_ROUGH2_VFV_01(i_xExtIlkOK := TMO_ROUGH1_VRC_01.M_IsClosed() AND TMO_ROUGH2_VRC_01.M_IsClosed()AND MR3K4_KBO_VWC_01.M_IsClosed() AND LI3K4_IP1_VWC_01.M_IsClosed());
ELSIF (IP1_ROUGH_VRC_02_AtOpnLS )THEN // vent entire end station
     TMO_ROUGH2_VFV_01(i_xExtIlkOK := TMO_ROUGH1_VRC_01.M_IsClosed() AND TMO_ROUGH2_VRC_01.M_IsClosed()AND MR3K4_KBO_VWC_01.M_IsClosed() AND LI3K4_IP1_VWC_01.M_IsClosed());
    ELSE //vent part of the IP1 when IP1_ROUGH_VRC_02 is not open
     TMO_ROUGH2_VFV_01(i_xExtIlkOK := TMO_ROUGH2_VRC_01.M_IsClosed());
END_IF

//MR5K4 and TM2K4 Inteface with DREAM
//Close window valve from DREAM PLC
IF bCLOSE_TMO_MR5K4_VWC THEN
    MR5K4_KBO_VWC_01.M_Set_OPN_SW(FALSE);
END_IF

IF bCLOSE_TMO_TM2K4_VWC THEN
    TM2K4_KBO_VWC_01.M_Set_OPN_SW(FALSE);
END_IF

//Send innformation about limit switch to DREAM PLC
bTMO_MR5K4_VWC_CLOSED_LS := MR5K4_KBO_VWC_01.iq_stValve.i_xClsLS;
bTMO_TM2K4_VWC_CLOSED_LS := TM2K4_KBO_VWC_01.iq_stValve.i_xClsLS;
bTMO_MR5K4_VWC_OPEN_LS	:= MR5K4_KBO_VWC_01.iq_stValve.i_xOpnLS;
bTMO_TM2K4_VWC_OPEN_LS	:= TM2K4_KBO_VWC_01.iq_stValve.i_xOpnLS;

END_PROGRAM

// ---- POUs/PRG_Roughing_Pumps.TcPOU
PROGRAM PRG_Roughing_Pumps
VAR

    xRough1Vrc01_OpenOK: BOOL := False;
    xRough1Vrc02_OpenOK: BOOL := False;
    xRough2Vrc01_OpenOK: BOOL := False;
    dummy_FFFO : FB_HardwareFFOutput;
    dummy_fbArbiter1    :   FB_Arbiter(1);

    PA1K4_IP1_PTM_01_xExtIlkOK: BOOL := FALSE;
    PA1K4_IP1_PTM_02_xExtIlkOK: BOOL := FALSE;
    PA1K4_IP1_PTM_03_xExtIlkOK: BOOL := False;

    f_trig_r1 : F_TRIG;
    f_trig_r2 : F_TRIG;
    r_trig_r1 : R_TRIG;
    r_trig_r2 : R_TRIG;

    tonDelOK : TON;
    tDelOK	:	TIME := T#30S;
    xExtIlkOK : BOOL;

    tonDelSW : TON;


    IM4K4_PPM_PTM_01_xExtIlkOK: BOOL := FALSE;
    LI1K4_IP1_PTM_01_xExtIlkOK: BOOL := FALSE;
    LI3K4_IP1_OUT_PTM_01_xExtIlkOK: BOOL := False;
    IM5K4_PPM_PTM_01_xExtIlkOK: BOOL := False;

    rTolerance : REAL;
    xDifPressureOK : BOOL := FALSE;
    TMO_ROUGH1_VRC_01_xExt_OK : BOOL;
    TMO_ROUGH1_VRC_02_xExt_OK : BOOL;
    TMO_ROUGH2_VRC_01_xExt_OK : BOOL;

    xLAMP_VRC01_VRC02_atOpnLS: BOOL;
END_VAR

VAR RETAIN
    TM1K4_PTM_01_xExtIlkOK: BOOL := False;
END_VAR


(* Roughing Valves *)

(* All three roughing valves permit to open when both side reading pressure below than setpoint, 1E-3 for both sides.
   When chamber is vented, bypass to open valve to pump down.
   FB_VGC_2S is used for VRC controls.

   For TMO_ROUGH1_VRC_01 & TMO_ROUGH1_VRC_02, additional interlock is implemented using i_xExt_OK input of VGC function:
   If pressure difference between TMO_ROUGH1_GPI_02 and TMO_ROUGH1_GPI_03 is greater than 20 Torr,
   only one of them permit to open.

   For TMO_ROUGH1_VRC_01 & TMO_ROUGH2_VRC_01 if one closed, wait for 10s, close the other.

*)


(* Check the pressure difference between TMO_ROUGH1_GPI_02 and TMO_ROUGH1_GPI_03 *)



rTolerance := 0.1;
xDifPressureOK := (ABS(TMO_ROUGH1_GPI_02.PG.rPRESS - TMO_ROUGH1_GPI_03.PG.rPRESS ) <= rTolerance ) AND
                  TMO_ROUGH1_GPI_02.PG.xPRESS_OK AND TMO_ROUGH1_GPI_03.PG.xPRESS_OK;

(* Set Rough1_vrc_01 external interlock OK TRUE, when:
     xDifPressureOK or TMO_ROUGH1_VRC_02 is closed
     AND if LAMP is connected, LAMP_ROUGH_VRC01 and VRC02 are open OR TMO_ROUGH2_VRC01 is open. *)

//IP1_ECAT_COM_ERROR = TRUE means that there is an EtherCAT Bridge Communication error.
IP1_ECAT_COM_ERROR := (xEcatBridge_TxPDO_state OR xEcatBridge_External_device_not_connected OR xEcatBridge_WcState);

xLAMP_VRC01_VRC02_atOpnLS := IP1_ROUGH_VRC_01_AtOpnLS AND NOT IP1_ECAT_COM_ERROR
                              AND IP1_ROUGH_VRC_02_AtOpnLS AND NOT IP1_ECAT_COM_ERROR;

//removing interlock from tmo_rough2_vrc_01 and IP1_VRC_02 interlock per James' request on 10-04-24
TMO_ROUGH1_VRC_01_xExt_OK := ( xDifPressureOK OR TMO_ROUGH1_VRC_02.iq_stValve.i_xClsLS )
                            AND (
                                  (IP1_ROUGH_VRC_01_AtOpnLS
                                  AND NOT IP1_ECAT_COM_ERROR)
                                  OR xPipe_replace_IP1  //request by Jeff on 8-21-25 to bypass ip1 logic when pipe is in

                               (*   and TMO_ROUGH2_VRC_01.iq_stValve.i_xOpnLS
                                  OR xLAMP_VRC01_VRC02_atOpnLS *)
                                 );


(* Set external interlock OK TRUE, when xDifPressureOK or TMO_ROUGH1_VRC_01 is closed *)

TMO_ROUGH1_VRC_02_xExt_OK := xDifPressureOK  OR TMO_ROUGH1_VRC_01.iq_stValve.i_xClsLS;
//make override of tmo_rough1_vrc-01 simple on 10-04-24

TMO_ROUGH1_VRC_01(
                i_stUSG := TMO_ROUGH1_GPI_02.PG,
                i_stDSG:= TMO_ROUGH1_GPI_01.PG,
                i_xDis_DPIlk := FALSE,
                i_xEPS_OK := TRUE,
                i_xPMPS_OK := TRUE,
                i_xExt_OK := TMO_ROUGH1_VRC_01_xExt_OK,
                i_xOverrideMode := xSystemOverrideMode_TMO AND xDifPressureOK(*TMO_ROUGH1_VRC_01_xExt_OK *),
                i_xReset := False,
                io_fbFFHWO :=dummy_FFFO,
                fbArbiter := dummy_fbArbiter1,
);


//make override of tmo_rough1_vrc-02 simple on 10-04-24

TMO_ROUGH1_VRC_02(
                i_stUSG := TMO_ROUGH1_GPI_03.PG,
                i_stDSG:= TMO_ROUGH1_GPI_01.PG,
                i_xDis_DPIlk := FALSE,
                i_xEPS_OK := TRUE,
                i_xPMPS_OK := TRUE,
                i_xExt_OK := TMO_ROUGH1_VRC_02_xExt_OK,
                i_xOverrideMode := xSystemOverrideMode_TMO AND xDifPressureOK (*TMO_ROUGH1_VRC_02_xExt_OK*),
                i_xReset := false,
                io_fbFFHWO :=dummy_FFFO,
                fbArbiter := dummy_fbArbiter1);


(* Set TMO_ROUGH2_VRC01 external interlock OK TRUE, if LAMP is connected, and either LAMP_ROUGH_VRC01, VRC02 and VRC03 are open
                    or both TMO_ROUGH1_VRC_01 and lamp_rough_vrc03 are open*)
//remove interlock with tmo_rough1_vrc_01 and IP1_rough_vrc_02, 01 and 03 interlocks per James's request on 10-04-24
TMO_ROUGH2_VRC_01_xExt_OK := (NOT IP1_ECAT_COM_ERROR AND
                        (  (IP1_ROUGH_VRC_01_AtOpnLS AND NOT IP1_ECAT_COM_ERROR
                                                  (*      AND IP1_ROUGH_VRC_02_AtOpnLS AND NOT IP1_ECAT_COM_ERROR *)
                                                        AND IP1_ROUGH_VRC_03_AtOpnLS AND NOT IP1_ECAT_COM_ERROR )
                        (*  OR ( TMO_ROUGH1_VRC_01.iq_stValve.i_xOpnLS and IP1_ROUGH_VRC_03_AtOpnLS AND NOT IP1_ECAT_COM_ERROR) *)
                          )) OR xPipe_replace_IP1 ;  //requested by jeff to use pipe to replace IP1 08-21-25

TMO_ROUGH2_VRC_01(
                i_stUSG := TMO_ROUGH2_GPI_02.PG,
                i_stDSG:= TMO_ROUGH2_GPI_01.PG,
                i_xDis_DPIlk := FALSE,
                i_xEPS_OK := TRUE,
                i_xPMPS_OK := TRUE,
                i_xExt_OK := TMO_ROUGH2_VRC_01_xExt_OK,
                i_xOverrideMode := xSystemOverrideMode_TMO,
                i_xReset := false,
                io_fbFFHWO :=dummy_FFFO,
                fbArbiter := dummy_fbArbiter1);




(* Granite 1 K4S2 Differential Turbo pumps *)


(* check if PA1K4_IP1_PTM_03 is Atspd, if it is starting, set up a timer for 30s to *)

xExtIlkOK := F_Turbo_Protection_ILK(i_stTurbo := PA1K4_IP1_PTM_01.iq_stPTM,
            i_stISG := TMO_ROUGH1_GPI_02.PG,
            i_stBSG := TMO_ROUGH1_GPI_02.PG,
            iq_stValve := TMO_ROUGH1_VRC_01.iq_stValve)	;

(* start when PTM03 is on*)
IF (PA1K4_IP1_PTM_03.iq_stPTM.i_xAtSpd) AND (NOT PA1K4_IP1_PTM_03.iq_stPTM.i_xFault) THEN
        PA1K4_IP1_PTM_01_xExtIlkOK := xExtIlkOK;

ELSIF (PA1K4_IP1_PTM_03.iq_stPTM.q_RunDO ) AND (NOT PA1K4_IP1_PTM_03.iq_stPTM.i_xFault ) THEN
    //delay timer
//  	  tonDelOK(IN:= xExtIlkOK, PT:=tDelOK);
    PA1K4_IP1_PTM_01_xExtIlkOK := xExtIlkOK ;
ELSE
        PA1K4_IP1_PTM_01_xExtIlkOK := FALSE;
END_IF


xExtIlkOK := F_Turbo_Protection_ILK(i_stTurbo := PA1K4_IP1_PTM_02.iq_stPTM,
            i_stISG := TMO_ROUGH1_GPI_02.PG,
            i_stBSG := TMO_ROUGH1_GPI_02.PG,
            iq_stValve := TMO_ROUGH1_VRC_01.iq_stValve)	;

IF (PA1K4_IP1_PTM_03.iq_stPTM.i_xAtSpd) AND (NOT PA1K4_IP1_PTM_03.iq_stPTM.i_xFault) THEN
        PA1K4_IP1_PTM_02_xExtIlkOK := xExtIlkOK;

ELSIF (PA1K4_IP1_PTM_03.iq_stPTM.q_RunDO ) AND (NOT PA1K4_IP1_PTM_03.iq_stPTM.i_xFault ) THEN
    //delay timer
//  	  tonDelOK(IN:= xExtIlkOK, PT:=tDelOK);
    PA1K4_IP1_PTM_02_xExtIlkOK := xExtIlkOK;
ELSE
        PA1K4_IP1_PTM_02_xExtIlkOK := FALSE;
END_IF

PA1K4_IP1_PTM_03_xExtIlkOK  := F_Turbo_Protection_ILK(i_stTurbo := PA1K4_IP1_PTM_03.iq_stPTM,
            i_stISG := TMO_ROUGH1_GPI_02.PG,
            i_stBSG := TMO_ROUGH1_GPI_02.PG,
            iq_stValve := TMO_ROUGH1_VRC_01.iq_stValve)	;


PA1K4_IP1_PTM_01(i_xExtIlkOK := PA1K4_IP1_PTM_01_xExtIlkOK , iq_stPTM => );

PA1K4_IP1_PTM_02(i_xExtIlkOK := PA1K4_IP1_PTM_02_xExtIlkOK, iq_stPTM => );
PA1K4_IP1_PTM_03(i_xExtIlkOK := PA1K4_IP1_PTM_03_xExtIlkOK, iq_stPTM => );

(*Serial Interface*)
(*Assign adresses to the pfeiffer controllers connected to this serial terminal*)
st_Pfeiffer_CTRL_PTM_01_02_03[1].iSerialAddress :=10;//PA1K4_IP1_PTM_01
st_Pfeiffer_CTRL_PTM_01_02_03[1].xEnableComm := TRUE;
st_Pfeiffer_CTRL_PTM_01_02_03[2].iSerialAddress :=9;//PA1K4_IP1_PTM_02
st_Pfeiffer_CTRL_PTM_01_02_03[2].xEnableComm := TRUE;
st_Pfeiffer_CTRL_PTM_01_02_03[3].iSerialAddress :=1;//PA1K4_IP1_PTM_03
st_Pfeiffer_CTRL_PTM_01_02_03[3].xEnableComm := TRUE;
(* Instanitate the Function block for serial communication with Pfeiffer*)
PA1K4_IP1_PTM_01_02_03_COM(astPfeifferControl := st_Pfeiffer_CTRL_PTM_01_02_03,
               astPfeifferStatus:= st_Pfeiffer_RBK_PTM_01_02_03,
                SerialRXBuffer:= K4S2_02_E10_SerialRXBuffer,
                SerialTXBuffer:= K4S2_02_E10_SerialTXBuffer);
(* Copy Status Pv's into the PTM structure*)
PA1K4_IP1_PTM_01.M_Serial_IO(st_Pfeiffer_CTRL:=st_Pfeiffer_CTRL_PTM_01_02_03[1],st_Pfeiffer_RBK:=st_Pfeiffer_RBK_PTM_01_02_03[1]);
PA1K4_IP1_PTM_02.M_Serial_IO(st_Pfeiffer_CTRL:=st_Pfeiffer_CTRL_PTM_01_02_03[2],st_Pfeiffer_RBK:=st_Pfeiffer_RBK_PTM_01_02_03[2]);
PA1K4_IP1_PTM_03.M_Serial_IO(st_Pfeiffer_CTRL:=st_Pfeiffer_CTRL_PTM_01_02_03[3],st_Pfeiffer_RBK:=st_Pfeiffer_RBK_PTM_01_02_03[3]);

(* Leybold turbo pumps on Granite 1 *)

IM4K4_PPM_PTM_01_xExtIlkOK := F_Turbo_Protection_ILK(i_stTurbo := IM4K4_PPM_PTM_01.iq_stPTM,
            i_stISG := TMO_ROUGH1_GPI_02.PG,
            i_stBSG := TMO_ROUGH1_GPI_02.PG,
            iq_stValve := TMO_ROUGH1_VRC_01.iq_stValve)	;

IM4K4_PPM_PTM_01(i_xExtIlkOK := IM4K4_PPM_PTM_01_xExtIlkOK, iq_stPTM => );



(* Instanitate the Function block for serial communication with TD20 *)
IM4K4_PPM_PTM_01_COM(SerialRXBuffer := K4S2_02_E17_SerialRXBuffer,
                SerialTXBuffer:= K4S2_02_E17_SerialTXBuffer,
                astTD20Status=>);
(* Copy Status Pv's into the PTM structure*)
IM4K4_PPM_PTM_01.M_Serial_IO(IM4K4_PPM_PTM_01_COM.astTD20Status);



LI1K4_IP1_PTM_01_xExtIlkOK := F_Turbo_Protection_ILK(i_stTurbo := LI1K4_IP1_PTM_01.iq_stPTM,
            i_stISG := TMO_ROUGH1_GPI_02.PG,
            i_stBSG := TMO_ROUGH1_GPI_02.PG,
            iq_stValve := TMO_ROUGH1_VRC_01.iq_stValve)	;

LI1K4_IP1_PTM_01(i_xExtIlkOK := LI1K4_IP1_PTM_01_xExtIlkOK, iq_stPTM => );

(* Instanitate the Function block for serial communication with TD20 *)
LI1K4_IP1_PTM_01_COM(SerialRXBuffer := K4S2_02_E18_SerialRXBuffer,
                SerialTXBuffer:= K4S2_02_E18_SerialTXBuffer,
                astTD20Status=>);
(* Copy Status Pv's into the PTM structure*)
LI1K4_IP1_PTM_01.M_Serial_IO(LI1K4_IP1_PTM_01_COM.astTD20Status);



(* Granite 2 K4S6 *)

LI3K4_IP1_OUT_PTM_01_xExtIlkOK := F_Turbo_Protection_ILK(i_stTurbo := LI3K4_IP1_OUT_PTM_01.iq_stPTM,
            i_stISG := PA2K4_IP1_GPI_01.PG,
            i_stBSG := TMO_ROUGH1_GPI_03.PG,
            iq_stValve := TMO_ROUGH1_VRC_02.iq_stValve)	;

LI3K4_IP1_OUT_PTM_01(i_xExtIlkOK := LI3K4_IP1_OUT_PTM_01_xExtIlkOK, iq_stPTM => );

TM1K4_PTM_01_xExtIlkOK := F_Turbo_Protection_ILK(i_stTurbo := TM1K4_PTM_01.iq_stPTM,
            i_stISG := PA2K4_IP1_GPI_01.PG,
            i_stBSG := TMO_ROUGH1_GPI_03.PG,
            iq_stValve := TMO_ROUGH1_VRC_02.iq_stValve)	;

TM1K4_PTM_01(i_xExtIlkOK := TM1K4_PTM_01_xExtIlkOK, iq_stPTM => );

IM5K4_PPM_PTM_01_xExtIlkOK := F_Turbo_Protection_ILK(i_stTurbo := IM5K4_PPM_PTM_01.iq_stPTM,
            i_stISG := PA2K4_IP1_GPI_01.PG,
            i_stBSG := TMO_ROUGH1_GPI_03.PG,
            iq_stValve := TMO_ROUGH1_VRC_02.iq_stValve)	;

IM5K4_PPM_PTM_01(i_xExtIlkOK := IM5K4_PPM_PTM_01_xExtIlkOK, iq_stPTM => );

(*Serial Interface*)
(*Assign adresses to the pfeiffer controllers connected to this serial terminal*)
st_Pfeiffer_CTRL_PTM_Granite2[1].iSerialAddress :=1;//LI3K4_IP1_OUT_PTM_01
st_Pfeiffer_CTRL_PTM_Granite2[1].xEnableComm := TRUE;
st_Pfeiffer_CTRL_PTM_Granite2[2].iSerialAddress :=7;//TM1K4_PTM_01
st_Pfeiffer_CTRL_PTM_Granite2[2].xEnableComm := TRUE;
st_Pfeiffer_CTRL_PTM_Granite2[3].iSerialAddress :=9; //IM5K4_PPM_PTM_01
st_Pfeiffer_CTRL_PTM_Granite2[3].xEnableComm := TRUE;
(* Instanitate the Function block for serial communication with Pfeiffer*)
Granite2_PTM_COM(astPfeifferControl := st_Pfeiffer_CTRL_PTM_Granite2,
               astPfeifferStatus:= st_Pfeiffer_RBK_PTM_Granite2,
                SerialRXBuffer:= K4S6_01_E5_SerialRXBuffer,
                SerialTXBuffer:= K4S6_01_E5_SerialTXBuffer);
(* Copy Status Pv's into the PTM structure*)
LI3K4_IP1_OUT_PTM_01.M_Serial_IO(st_Pfeiffer_CTRL:=st_Pfeiffer_CTRL_PTM_Granite2[1],st_Pfeiffer_RBK:=st_Pfeiffer_RBK_PTM_Granite2[1]);
TM1K4_PTM_01.M_Serial_IO(st_Pfeiffer_CTRL:=st_Pfeiffer_CTRL_PTM_Granite2[2],st_Pfeiffer_RBK:=st_Pfeiffer_RBK_PTM_Granite2[2]);
IM5K4_PPM_PTM_01.M_Serial_IO(st_Pfeiffer_CTRL:=st_Pfeiffer_CTRL_PTM_Granite2[3],st_Pfeiffer_RBK:=st_Pfeiffer_RBK_PTM_Granite2[3]);

END_PROGRAM
